  MoveL 9971 to (-27.77, 164.22, 135.08) mm, rotated rx 180 ry 0 rz 180 deg; joints [-126.617, -52.338, -80.882, 63.029, 64.237, -40.501]
  Call Extruder(390.70034)
  MoveL 9972 to (-28.02, 164.17, 135.08) mm, rotated rx 180 ry 0 rz 180 deg; joints [-126.595, -52.322, -80.919, 63.038, 64.26, -40.489]
  MoveL 9973 to (-28.02, 164.17, 135.08) mm, rotated rx 180 ry 0 rz 180 deg; joints [-126.595, -52.322, -80.919, 63.038, 64.26, -40.489]
  Call Extruder(390.83670)
  MoveL 9974 to (-28.27, 164.12, 135.08) mm, rotated rx 180 ry 0 rz -180 deg; joints [-126.573, -52.305, -80.957, 63.048, 64.284, -40.477]
  MoveL 9975 to (-28.27, 164.12, 135.08) mm, rotated rx 180 ry 0 rz -180 deg; joints [-126.573, -52.305, -80.957, 63.048, 64.284, -40.477]
  Call Extruder(390.97368)
  MoveL 9976 to (-28.52, 164.07, 135.08) mm, rotated rx 180 ry 0 rz 180 deg; joints [-126.551, -52.288, -80.994, 63.058, 64.307, -40.464]
  MoveL 9977 to (-28.52, 164.07, 135.08) mm, rotated rx 180 ry 0 rz 180 deg; joints [-126.551, -52.288, -80.994, 63.058, 64.307, -40.464]
  Call Extruder(391.11127)
  MoveL 9978 to (-28.77, 164.02, 135.08) mm, rotated rx -180 ry 0 rz 180 deg; joints [-126.529, -52.272, -81.031, 63.067, 64.331, -40.452]
  MoveL 9979 to (-28.77, 164.02, 135.08) mm, rotated rx -180 ry 0 rz 180 deg; joints [-126.529, -52.272, -81.031, 63.067, 64.331, -40.452]
  Call Extruder(391.22498)
  MoveL 9980 to (-28.97, 163.97, 135.08) mm, rotated rx 180 ry 0 rz 180 deg; joints [-126.511, -52.258, -81.062, 63.075, 64.35, -40.441]
  MoveL 9981 to (-28.97, 163.97, 135.08) mm, rotated rx 180 ry 0 rz 180 deg; joints [-126.511, -52.258, -81.062, 63.075, 64.35, -40.441]
  Call Extruder(391.33915)
  MoveL 9982 to (-29.18, 163.93, 135.08) mm, rotated rx 180 ry 0 rz 180 deg; joints [-126.494, -52.244, -81.093, 63.082, 64.369, -40.431]
  MoveL 9983 to (-29.18, 163.93, 135.08) mm, rotated rx 180 ry 0 rz 180 deg; joints [-126.494, -52.244, -81.093, 63.082, 64.369, -40.431]
  Call Extruder(391.45377)
  MoveL 9984 to (-29.38, 163.88, 135.08) mm, rotated rx -180 ry 0 rz 180 deg; joints [-126.476, -52.23, -81.125, 63.09, 64.389, -40.42]
  MoveL 9985 to (-29.38, 163.88, 135.08) mm, rotated rx -180 ry 0 rz 180 deg; joints [-126.476, -52.23, -81.125, 63.09, 64.389, -40.42]
  Call Extruder(391.56884)
  MoveL 9986 to (-29.59, 163.84, 135.08) mm, rotated rx 180 ry 0 rz 180 deg; joints [-126.459, -52.216, -81.155, 63.098, 64.408, -40.41]
  MoveL 9987 to (-29.59, 163.84, 135.08) mm, rotated rx 180 ry 0 rz 180 deg; joints [-126.459, -52.216, -81.155, 63.098, 64.408, -40.41]
  Call Extruder(391.69108)
  MoveL 9988 to (-29.8, 163.78, 135.08) mm, rotated rx -180 ry 0 rz 180 deg; joints [-126.441, -52.201, -81.189, 63.105, 64.428, -40.397]
  MoveL 9989 to (-29.8, 163.78, 135.08) mm, rotated rx -180 ry 0 rz 180 deg; joints [-126.441, -52.201, -81.189, 63.105, 64.428, -40.397]
  Call Extruder(391.82075)
  MoveL 9990 to (-30.02, 163.72, 135.08) mm, rotated rx -180 ry 0 rz 180 deg; joints [-126.423, -52.184, -81.227, 63.111, 64.449, -40.384]
  MoveL 9991 to (-30.02, 163.72, 135.08) mm, rotated rx -180 ry 0 rz 180 deg; joints [-126.423, -52.184, -81.227, 63.111, 64.449, -40.384]
  Call Extruder(391.95100)
  MoveL 9992 to (-30.25, 163.65, 135.08) mm, rotated rx 180 ry 0 rz 180 deg; joints [-126.405, -52.168, -81.263, 63.117, 64.47, -40.37]
  MoveL 9993 to (-30.25, 163.65, 135.08) mm, rotated rx 180 ry 0 rz 180 deg; joints [-126.405, -52.168, -81.263, 63.117, 64.47, -40.37]
  Call Extruder(392.08180)
  MoveL 9994 to (-30.47, 163.58, 135.08) mm, rotated rx 180 ry 0 rz 180 deg; joints [-126.387, -52.151, -81.3, 63.124, 64.491, -40.356]
  MoveL 9995 to (-30.47, 163.58, 135.08) mm, rotated rx 180 ry 0 rz 180 deg; joints [-126.387, -52.151, -81.3, 63.124, 64.491, -40.356]
  Call Extruder(392.21318)
  MoveL 9996 to (-30.69, 163.51, 135.08) mm, rotated rx 180 ry 0 rz 180 deg; joints [-126.369, -52.135, -81.337, 63.13, 64.512, -40.343]
  MoveL 9997 to (-30.69, 163.51, 135.08) mm, rotated rx 180 ry 0 rz 180 deg; joints [-126.369, -52.135, -81.337, 63.13, 64.512, -40.343]
  Call Extruder(392.32507)
  MoveL 9998 to (-30.88, 163.45, 135.08) mm, rotated rx 180 ry 0 rz 180 deg; joints [-126.354, -52.121, -81.369, 63.135, 64.529, -40.331]
  MoveL 9999 to (-30.88, 163.45, 135.08) mm, rotated rx 180 ry 0 rz 180 deg; joints [-126.354, -52.121, -81.369, 63.135, 64.529, -40.331]
  Call Extruder(392.43740)
  MoveL 10000 to (-31.07, 163.39, 135.08) mm, rotated rx 180 ry 0 rz 180 deg; joints [-126.339, -52.107, -81.401, 63.141, 64.547, -40.319]
  MoveL 10001 to (-31.07, 163.39, 135.08) mm, rotated rx 180 ry 0 rz 180 deg; joints [-126.339, -52.107, -81.401, 63.141, 64.547, -40.319]
  Call Extruder(392.55019)
  MoveL 10002 to (-31.26, 163.33, 135.08) mm, rotated rx 180 ry 0 rz 180 deg; joints [-126.324, -52.092, -81.433, 63.146, 64.564, -40.307]
  MoveL 10003 to (-31.26, 163.33, 135.08) mm, rotated rx 180 ry 0 rz 180 deg; joints [-126.324, -52.092, -81.433, 63.146, 64.564, -40.307]
  Call Extruder(392.66341)
  MoveL 10004 to (-31.45, 163.27, 135.08) mm, rotated rx -180 ry 0 rz -180 deg; joints [-126.309, -52.078, -81.464, 63.151, 64.582, -40.295]
  MoveL 10005 to (-31.45, 163.27, 135.08) mm, rotated rx -180 ry 0 rz -180 deg; joints [-126.309, -52.078, -81.464, 63.151, 64.582, -40.295]
  Call Extruder(392.77708)
  MoveL 10006 to (-31.64, 163.21, 135.08) mm, rotated rx 180 ry 0 rz 180 deg; joints [-126.294, -52.064, -81.496, 63.156, 64.599, -40.283]
  MoveL 10007 to (-31.64, 163.21, 135.08) mm, rotated rx 180 ry 0 rz 180 deg; joints [-126.294, -52.064, -81.496, 63.156, 64.599, -40.283]
  Call Extruder(392.95906)
  MoveL 10008 to (-31.93, 163.09, 135.08) mm, rotated rx 180 ry 0 rz 180 deg; joints [-126.273, -52.041, -81.549, 63.161, 64.626, -40.261]
  MoveL 10009 to (-31.93, 163.09, 135.08) mm, rotated rx 180 ry 0 rz 180 deg; joints [-126.273, -52.041, -81.549, 63.161, 64.626, -40.261]
  Call Extruder(393.14179)
  MoveL 10010 to (-32.22, 162.96, 135.08) mm, rotated rx -180 ry 0 rz -180 deg; joints [-126.252, -52.017, -81.602, 63.167, 64.653, -40.24]
  MoveL 10011 to (-32.22, 162.96, 135.08) mm, rotated rx -180 ry 0 rz -180 deg; joints [-126.252, -52.017, -81.602, 63.167, 64.653, -40.24]
  Call Extruder(393.31221)
  MoveL 10012 to (-32.49, 162.85, 135.08) mm, rotated rx 180 ry 0 rz -180 deg; joints [-126.233, -51.995, -81.652, 63.171, 64.678, -40.22]
  MoveL 10013 to (-32.49, 162.85, 135.08) mm, rotated rx 180 ry 0 rz -180 deg; joints [-126.233, -51.995, -81.652, 63.171, 64.678, -40.22]
  Call Extruder(393.47018)
  MoveL 10014 to (-32.74, 162.74, 135.08) mm, rotated rx -180 ry 0 rz 180 deg; joints [-126.215, -51.974, -81.698, 63.176, 64.701, -40.201]
  MoveL 10015 to (-32.74, 162.74, 135.08) mm, rotated rx -180 ry 0 rz 180 deg; joints [-126.215, -51.974, -81.698, 63.176, 64.701, -40.201]
  Call Extruder(393.62876)
  MoveL 10016 to (-32.99, 162.64, 135.08) mm, rotated rx 180 ry 0 rz 180 deg; joints [-126.197, -51.954, -81.744, 63.18, 64.724, -40.182]
  MoveL 10017 to (-32.99, 162.64, 135.08) mm, rotated rx 180 ry 0 rz 180 deg; joints [-126.197, -51.954, -81.744, 63.18, 64.724, -40.182]
  Call Extruder(393.83493)
  MoveL 10018 to (-33.29, 162.46, 135.08) mm, rotated rx 180 ry 0 rz 180 deg; joints [-126.179, -51.926, -81.807, 63.181, 64.752, -40.154]
  MoveL 10019 to (-33.29, 162.46, 135.08) mm, rotated rx 180 ry 0 rz 180 deg; joints [-126.179, -51.926, -81.807, 63.181, 64.752, -40.154]
  Call Extruder(394.04187)
  MoveL 10020 to (-33.6, 162.29, 135.08) mm, rotated rx 180 ry 0 rz -180 deg; joints [-126.16, -51.898, -81.87, 63.182, 64.78, -40.126]
  MoveL 10021 to (-33.6, 162.29, 135.08) mm, rotated rx 180 ry 0 rz -180 deg; joints [-126.16, -51.898, -81.87, 63.182, 64.78, -40.126]
  Call Extruder(394.24959)
  MoveL 10022 to (-33.9, 162.11, 135.08) mm, rotated rx 180 ry 0 rz -180 deg; joints [-126.142, -51.87, -81.933, 63.183, 64.807, -40.099]
  MoveL 10023 to (-33.9, 162.11, 135.08) mm, rotated rx 180 ry 0 rz -180 deg; joints [-126.142, -51.87, -81.933, 63.183, 64.807, -40.099]
  Call Extruder(394.45809)
  MoveL 10024 to (-34.21, 161.94, 135.08) mm, rotated rx 180 ry 0 rz -180 deg; joints [-126.123, -51.842, -81.996, 63.183, 64.835, -40.071]
  MoveL 10025 to (-34.21, 161.94, 135.08) mm, rotated rx 180 ry 0 rz -180 deg; joints [-126.123, -51.842, -81.996, 63.183, 64.835, -40.071]
  Call Extruder(394.63764)
  MoveL 10026 to (-34.45, 161.76, 135.08) mm, rotated rx 180 ry 0 rz 180 deg; joints [-126.111, -51.817, -82.052, 63.181, 64.857, -40.044]
  MoveL 10027 to (-34.45, 161.76, 135.08) mm, rotated rx 180 ry 0 rz 180 deg; joints [-126.111, -51.817, -82.052, 63.181, 64.857, -40.044]
  Call Extruder(394.97107)
  MoveL 10028 to (-34.9, 161.43, 135.08) mm, rotated rx 180 ry 0 rz 180 deg; joints [-126.089, -51.77, -82.156, 63.175, 64.897, -39.995]
  MoveL 10029 to (-34.9, 161.43, 135.08) mm, rotated rx 180 ry 0 rz 180 deg; joints [-126.089, -51.77, -82.156, 63.175, 64.897, -39.995]
  Call Extruder(395.30569)
  MoveL 10030 to (-35.35, 161.1, 135.08) mm, rotated rx 180 ry 0 rz 180 deg; joints [-126.067, -51.724, -82.26, 63.17, 64.938, -39.946]
  Call Extruder(396.13360)
  MoveL 10031 to (-36.39, 160.19, 135.08) mm, rotated rx 180 ry 0 rz 180 deg; joints [-126.027, -51.607, -82.524, 63.142, 65.029, -39.816]
  Call Extruder(396.96153)
  MoveL 10032 to (-37.3, 159.15, 135.08) mm, rotated rx -180 ry 0 rz 180 deg; joints [-126.011, -51.488, -82.792, 63.095, 65.107, -39.675]
  Call Extruder(397.12884)
  MoveL 10033 to (-37.47, 158.93, 135.08) mm, rotated rx 180 ry 0 rz 180 deg; joints [-126.011, -51.464, -82.846, 63.082, 65.121, -39.646]
  MoveL 10034 to (-37.47, 158.93, 135.08) mm, rotated rx 180 ry 0 rz 180 deg; joints [-126.011, -51.464, -82.846, 63.082, 65.121, -39.646]
  Call Extruder(397.46227)
  MoveL 10035 to (-37.79, 158.48, 135.08) mm, rotated rx -180 ry 0 rz -180 deg; joints [-126.011, -51.416, -82.955, 63.057, 65.148, -39.586]
  MoveL 10036 to (-37.79, 158.48, 135.08) mm, rotated rx -180 ry 0 rz -180 deg; joints [-126.011, -51.416, -82.955, 63.057, 65.148, -39.586]
  Call Extruder(397.53291)
  MoveL 10037 to (-37.87, 158.38, 135.08) mm, rotated rx 180 ry 0 rz 180 deg; joints [-126.011, -51.406, -82.978, 63.052, 65.154, -39.573]
  Set speed (130.0 mm/s)
  MoveL 10038 to (-39.48, 155.51, 135.08) mm, rotated rx -180 ry 0 rz 180 deg; joints [-126.062, -51.125, -83.613, 62.863, 65.283, -39.207]
  MoveL 10039 to (-39.48, 155.51, 144.49) mm, rotated rx 180 ry 0 rz 180 deg; joints [-126.062, -49.882, -84.026, 63.207, 64.906, -40.024]
  MoveL 10040 to (-38.84, 156.79, 144.49) mm, rotated rx 180 ry 0 rz 180 deg; joints [-126.03, -50.005, -83.751, 63.296, 64.858, -40.184]
  Set speed (30.0 mm/s)
  MoveL 10041 to (-38.84, 156.79, 144.49) mm, rotated rx 180 ry 0 rz 180 deg; joints [-126.03, -50.005, -83.751, 63.296, 64.858, -40.184]
  Call Extruder(397.61221)
  MoveL 10042 to (-38.89, 156.66, 144.49) mm, rotated rx 180 ry 0 rz 180 deg; joints [-126.034, -49.994, -83.777, 63.287, 64.862, -40.169]
  MoveL 10043 to (-38.89, 156.66, 144.49) mm, rotated rx 180 ry 0 rz 180 deg; joints [-126.034, -49.994, -83.777, 63.287, 64.862, -40.169]
  Call Extruder(397.77019)
  MoveL 10044 to (-39, 156.42, 144.49) mm, rotated rx 180 ry 0 rz 180 deg; joints [-126.042, -49.971, -83.828, 63.268, 64.87, -40.138]
  MoveL 10045 to (-39, 156.42, 144.49) mm, rotated rx 180 ry 0 rz 180 deg; joints [-126.042, -49.971, -83.828, 63.268, 64.87, -40.138]
  Call Extruder(397.92758)
  MoveL 10046 to (-39.1, 156.17, 144.49) mm, rotated rx 180 ry 0 rz -180 deg; joints [-126.05, -49.948, -83.88, 63.25, 64.877, -40.107]
  MoveL 10047 to (-39.1, 156.17, 144.49) mm, rotated rx 180 ry 0 rz -180 deg; joints [-126.05, -49.948, -83.88, 63.25, 64.877, -40.107]
  Call Extruder(398.11030)
  MoveL 10048 to (-39.23, 155.88, 144.49) mm, rotated rx 180 ry 0 rz 180 deg; joints [-126.06, -49.921, -83.939, 63.228, 64.886, -40.072]
  MoveL 10049 to (-39.23, 155.88, 144.49) mm, rotated rx 180 ry 0 rz 180 deg; joints [-126.06, -49.921, -83.939, 63.228, 64.886, -40.072]
  Call Extruder(398.29226)
  MoveL 10050 to (-39.35, 155.58, 144.49) mm, rotated rx 180 ry 0 rz 180 deg; joints [-126.07, -49.894, -83.999, 63.206, 64.894, -40.036]
  MoveL 10051 to (-39.35, 155.58, 144.49) mm, rotated rx 180 ry 0 rz 180 deg; joints [-126.07, -49.894, -83.999, 63.206, 64.894, -40.036]
  Call Extruder(398.43959)
  MoveL 10052 to (-39.44, 155.34, 144.49) mm, rotated rx 180 ry 0 rz -180 deg; joints [-126.079, -49.872, -84.047, 63.187, 64.9, -40.007]
  MoveL 10053 to (-39.44, 155.34, 144.49) mm, rotated rx 180 ry 0 rz -180 deg; joints [-126.079, -49.872, -84.047, 63.187, 64.9, -40.007]
  Call Extruder(398.55283)
  MoveL 10054 to (-39.5, 155.15, 144.49) mm, rotated rx 180 ry 0 rz 180 deg; joints [-126.087, -49.856, -84.083, 63.172, 64.904, -39.984]
  MoveL 10055 to (-39.5, 155.15, 144.49) mm, rotated rx 180 ry 0 rz 180 deg; joints [-126.087, -49.856, -84.083, 63.172, 64.904, -39.984]
  Call Extruder(398.66562)
  MoveL 10056 to (-39.56, 154.97, 144.49) mm, rotated rx 180 ry 0 rz 180 deg; joints [-126.095, -49.839, -84.119, 63.157, 64.908, -39.962]
  MoveL 10057 to (-39.56, 154.97, 144.49) mm, rotated rx 180 ry 0 rz 180 deg; joints [-126.095, -49.839, -84.119, 63.157, 64.908, -39.962]
  Call Extruder(398.77796)
  MoveL 10058 to (-39.62, 154.78, 144.49) mm, rotated rx 180 ry 0 rz 180 deg; joints [-126.103, -49.823, -84.156, 63.142, 64.912, -39.939]
  MoveL 10059 to (-39.62, 154.78, 144.49) mm, rotated rx 180 ry 0 rz 180 deg; joints [-126.103, -49.823, -84.156, 63.142, 64.912, -39.939]
  Call Extruder(398.88986)
  MoveL 10060 to (-39.68, 154.59, 144.49) mm, rotated rx -180 ry 0 rz 180 deg; joints [-126.111, -49.806, -84.192, 63.126, 64.915, -39.916]
  MoveL 10061 to (-39.68, 154.59, 144.49) mm, rotated rx -180 ry 0 rz 180 deg; joints [-126.111, -49.806, -84.192, 63.126, 64.915, -39.916]
  Call Extruder(399.01126)
  MoveL 10062 to (-39.75, 154.38, 144.49) mm, rotated rx 180 ry 0 rz 180 deg; joints [-126.12, -49.789, -84.232, 63.11, 64.919, -39.892]
  MoveL 10063 to (-39.75, 154.38, 144.49) mm, rotated rx 180 ry 0 rz 180 deg; joints [-126.12, -49.789, -84.232, 63.11, 64.919, -39.892]
  Call Extruder(399.14206)
  MoveL 10064 to (-39.81, 154.16, 144.49) mm, rotated rx -180 ry 0 rz 180 deg; joints [-126.131, -49.769, -84.275, 63.091, 64.924, -39.865]
  MoveL 10065 to (-39.81, 154.16, 144.49) mm, rotated rx -180 ry 0 rz 180 deg; joints [-126.131, -49.769, -84.275, 63.091, 64.924, -39.865]
  Call Extruder(399.27229)
  MoveL 10066 to (-39.88, 153.94, 144.49) mm, rotated rx 180 ry 0 rz 180 deg; joints [-126.141, -49.75, -84.317, 63.073, 64.928, -39.838]
  MoveL 10067 to (-39.88, 153.94, 144.49) mm, rotated rx 180 ry 0 rz 180 deg; joints [-126.141, -49.75, -84.317, 63.073, 64.928, -39.838]
  Call Extruder(399.40195)
  MoveL 10068 to (-39.95, 153.71, 144.49) mm, rotated rx -180 ry 0 rz 180 deg; joints [-126.151, -49.731, -84.36, 63.054, 64.932, -39.811]
  MoveL 10069 to (-39.95, 153.71, 144.49) mm, rotated rx -180 ry 0 rz 180 deg; joints [-126.151, -49.731, -84.36, 63.054, 64.932, -39.811]
  Call Extruder(399.53105)
  MoveL 10070 to (-40.02, 153.49, 144.49) mm, rotated rx -180 ry 0 rz -180 deg; joints [-126.161, -49.712, -84.402, 63.036, 64.936, -39.785]
  MoveL 10071 to (-40.02, 153.49, 144.49) mm, rotated rx -180 ry 0 rz -180 deg; joints [-126.161, -49.712, -84.402, 63.036, 64.936, -39.785]
  Call Extruder(399.64614)
  MoveL 10072 to (-40.06, 153.28, 144.49) mm, rotated rx -180 ry 0 rz 180 deg; joints [-126.173, -49.695, -84.439, 63.018, 64.938, -39.761]
  MoveL 10073 to (-40.06, 153.28, 144.49) mm, rotated rx -180 ry 0 rz 180 deg; joints [-126.173, -49.695, -84.439, 63.018, 64.938, -39.761]
  Call Extruder(399.76077)
  MoveL 10074 to (-40.11, 153.08, 144.49) mm, rotated rx 180 ry 0 rz -180 deg; joints [-126.184, -49.679, -84.476, 63, 64.94, -39.737]
  MoveL 10075 to (-40.11, 153.08, 144.49) mm, rotated rx 180 ry 0 rz -180 deg; joints [-126.184, -49.679, -84.476, 63, 64.94, -39.737]
  Call Extruder(399.87495)
  MoveL 10076 to (-40.15, 152.88, 144.49) mm, rotated rx -180 ry 0 rz -180 deg; joints [-126.195, -49.662, -84.513, 62.982, 64.942, -39.713]
  MoveL 10077 to (-40.15, 152.88, 144.49) mm, rotated rx -180 ry 0 rz -180 deg; joints [-126.195, -49.662, -84.513, 62.982, 64.942, -39.713]
  Call Extruder(399.98868)
  MoveL 10078 to (-40.2, 152.67, 144.49) mm, rotated rx -180 ry 0 rz 180 deg; joints [-126.206, -49.645, -84.55, 62.964, 64.944, -39.689]
  MoveL 10079 to (-40.2, 152.67, 144.49) mm, rotated rx -180 ry 0 rz 180 deg; joints [-126.206, -49.645, -84.55, 62.964, 64.944, -39.689]
  Call Extruder(400.11411)
  MoveL 10080 to (-40.24, 152.45, 144.49) mm, rotated rx 180 ry 0 rz 180 deg; joints [-126.219, -49.627, -84.59, 62.944, 64.946, -39.662]
  MoveL 10081 to (-40.24, 152.45, 144.49) mm, rotated rx 180 ry 0 rz 180 deg; joints [-126.219, -49.627, -84.59, 62.944, 64.946, -39.662]
  Call Extruder(400.25109)
  MoveL 10082 to (-40.29, 152.2, 144.49) mm, rotated rx 180 ry 0 rz 180 deg; joints [-126.233, -49.607, -84.635, 62.921, 64.948, -39.633]
  MoveL 10083 to (-40.29, 152.2, 144.49) mm, rotated rx 180 ry 0 rz 180 deg; joints [-126.233, -49.607, -84.635, 62.921, 64.948, -39.633]
  Call Extruder(400.38745)
  MoveL 10084 to (-40.34, 151.95, 144.49) mm, rotated rx 180 ry 0 rz 180 deg; joints [-126.248, -49.587, -84.679, 62.899, 64.95, -39.604]
  MoveL 10085 to (-40.34, 151.95, 144.49) mm, rotated rx 180 ry 0 rz 180 deg; joints [-126.248, -49.587, -84.679, 62.899, 64.95, -39.604]
  Call Extruder(400.52321)
  MoveL 10086 to (-40.39, 151.7, 144.49) mm, rotated rx 180 ry 0 rz 180 deg; joints [-126.262, -49.567, -84.724, 62.877, 64.952, -39.575]
  MoveL 10087 to (-40.39, 151.7, 144.49) mm, rotated rx 180 ry 0 rz 180 deg; joints [-126.262, -49.567, -84.724, 62.877, 64.952, -39.575]
  Call Extruder(400.65835)
  MoveL 10088 to (-40.44, 151.45, 144.49) mm, rotated rx 180 ry 0 rz 180 deg; joints [-126.276, -49.547, -84.768, 62.854, 64.954, -39.546]
  MoveL 10089 to (-40.44, 151.45, 144.49) mm, rotated rx 180 ry 0 rz 180 deg; joints [-126.276, -49.547, -84.768, 62.854, 64.954, -39.546]
  Call Extruder(400.79289)
  MoveL 10090 to (-40.49, 151.2, 144.49) mm, rotated rx 180 ry 0 rz 180 deg; joints [-126.291, -49.527, -84.812, 62.832, 64.956, -39.517]
  MoveL 10091 to (-40.49, 151.2, 144.49) mm, rotated rx 180 ry 0 rz 180 deg; joints [-126.291, -49.527, -84.812, 62.832, 64.956, -39.517]
  Call Extruder(400.92681)
  MoveL 10092 to (-40.54, 150.95, 144.49) mm, rotated rx 180 ry 0 rz -180 deg; joints [-126.305, -49.508, -84.856, 62.81, 64.958, -39.487]
  MoveL 10093 to (-40.54, 150.95, 144.49) mm, rotated rx 180 ry 0 rz -180 deg; joints [-126.305, -49.508, -84.856, 62.81, 64.958, -39.487]
  Call Extruder(401.07467)
  MoveL 10094 to (-40.59, 150.67, 144.49) mm, rotated rx 180 ry 0 rz -180 deg; joints [-126.322, -49.486, -84.905, 62.784, 64.959, -39.455]
  MoveL 10095 to (-40.59, 150.67, 144.49) mm, rotated rx 180 ry 0 rz -180 deg; joints [-126.322, -49.486, -84.905, 62.784, 64.959, -39.455]
  Call Extruder(401.23639)
  MoveL 10096 to (-40.64, 150.37, 144.49) mm, rotated rx -180 ry 0 rz 180 deg; joints [-126.341, -49.462, -84.958, 62.756, 64.961, -39.42]
  MoveL 10097 to (-40.64, 150.37, 144.49) mm, rotated rx -180 ry 0 rz 180 deg; joints [-126.341, -49.462, -84.958, 62.756, 64.961, -39.42]
  Call Extruder(401.39739)
  MoveL 10098 to (-40.69, 150.06, 144.49) mm, rotated rx 180 ry 0 rz -180 deg; joints [-126.36, -49.438, -85.011, 62.728, 64.962, -39.384]
  MoveL 10099 to (-40.69, 150.06, 144.49) mm, rotated rx 180 ry 0 rz -180 deg; joints [-126.36, -49.438, -85.011, 62.728, 64.962, -39.384]
  Call Extruder(401.55766)
  MoveL 10100 to (-40.74, 149.76, 144.49) mm, rotated rx 180 ry 0 rz 180 deg; joints [-126.379, -49.415, -85.063, 62.7, 64.963, -39.349]
  MoveL 10101 to (-40.74, 149.76, 144.49) mm, rotated rx 180 ry 0 rz 180 deg; joints [-126.379, -49.415, -85.063, 62.7, 64.963, -39.349]
  Call Extruder(401.71721)
  MoveL 10102 to (-40.78, 149.45, 144.49) mm, rotated rx 180 ry 0 rz -180 deg; joints [-126.398, -49.391, -85.116, 62.671, 64.964, -39.314]
  MoveL 10103 to (-40.78, 149.45, 144.49) mm, rotated rx 180 ry 0 rz -180 deg; joints [-126.398, -49.391, -85.116, 62.671, 64.964, -39.314]
  Call Extruder(401.87602)
  MoveL 10104 to (-40.83, 149.14, 144.49) mm, rotated rx 180 ry 0 rz 180 deg; joints [-126.417, -49.367, -85.169, 62.643, 64.966, -39.278]
  MoveL 10105 to (-40.83, 149.14, 144.49) mm, rotated rx 180 ry 0 rz 180 deg; joints [-126.417, -49.367, -85.169, 62.643, 64.966, -39.278]
  Call Extruder(402.05468)
  MoveL 10106 to (-40.88, 148.8, 144.49) mm, rotated rx 180 ry 0 rz 180 deg; joints [-126.439, -49.341, -85.228, 62.61, 64.966, -39.238]
  MoveL 10107 to (-40.88, 148.8, 144.49) mm, rotated rx 180 ry 0 rz 180 deg; joints [-126.439, -49.341, -85.228, 62.61, 64.966, -39.238]
  Call Extruder(402.25313)
  MoveL 10108 to (-40.92, 148.41, 144.49) mm, rotated rx 180 ry 0 rz 180 deg; joints [-126.465, -49.312, -85.293, 62.573, 64.966, -39.194]
  MoveL 10109 to (-40.92, 148.41, 144.49) mm, rotated rx 180 ry 0 rz 180 deg; joints [-126.465, -49.312, -85.293, 62.573, 64.966, -39.194]
  Call Extruder(402.45070)
  MoveL 10110 to (-40.97, 148.02, 144.49) mm, rotated rx -180 ry 0 rz -180 deg; joints [-126.491, -49.282, -85.358, 62.536, 64.967, -39.149]
  MoveL 10111 to (-40.97, 148.02, 144.49) mm, rotated rx -180 ry 0 rz -180 deg; joints [-126.491, -49.282, -85.358, 62.536, 64.967, -39.149]
  Call Extruder(402.64741)
  MoveL 10112 to (-41.02, 147.63, 144.49) mm, rotated rx -180 ry 0 rz 180 deg; joints [-126.517, -49.253, -85.423, 62.499, 64.967, -39.105]
  MoveL 10113 to (-41.02, 147.63, 144.49) mm, rotated rx -180 ry 0 rz 180 deg; joints [-126.517, -49.253, -85.423, 62.499, 64.967, -39.105]
  Call Extruder(402.84324)
  MoveL 10114 to (-41.06, 147.25, 144.49) mm, rotated rx -180 ry 0 rz 180 deg; joints [-126.543, -49.224, -85.487, 62.462, 64.967, -39.06]
  MoveL 10115 to (-41.06, 147.25, 144.49) mm, rotated rx -180 ry 0 rz 180 deg; joints [-126.543, -49.224, -85.487, 62.462, 64.967, -39.06]
  Call Extruder(403.13864)
  MoveL 10116 to (-41.11, 146.66, 144.49) mm, rotated rx -180 ry 0 rz 180 deg; joints [-126.585, -49.181, -85.583, 62.404, 64.965, -38.993]
  MoveL 10117 to (-41.11, 146.66, 144.49) mm, rotated rx -180 ry 0 rz 180 deg; joints [-126.585, -49.181, -85.583, 62.404, 64.965, -38.993]
  Call Extruder(403.43270)
  MoveL 10118 to (-41.15, 146.07, 144.49) mm, rotated rx -180 ry 0 rz 180 deg; joints [-126.628, -49.138, -85.679, 62.345, 64.962, -38.926]
  MoveL 10119 to (-41.15, 146.07, 144.49) mm, rotated rx -180 ry 0 rz 180 deg; joints [-126.628, -49.138, -85.679, 62.345, 64.962, -38.926]
  Call Extruder(403.72544)
  MoveL 10120 to (-41.2, 145.48, 144.49) mm, rotated rx 180 ry 0 rz 180 deg; joints [-126.67, -49.096, -85.775, 62.287, 64.96, -38.859]
  MoveL 10121 to (-41.2, 145.48, 144.49) mm, rotated rx 180 ry 0 rz 180 deg; joints [-126.67, -49.096, -85.775, 62.287, 64.96, -38.859]
  Call Extruder(404.29889)
  MoveL 10122 to (-41.25, 144.32, 144.49) mm, rotated rx 180 ry 0 rz 180 deg; joints [-126.759, -49.014, -85.958, 62.169, 64.952, -38.728]
  MoveL 10123 to (-41.25, 144.32, 144.49) mm, rotated rx 180 ry 0 rz 180 deg; joints [-126.759, -49.014, -85.958, 62.169, 64.952, -38.728]
  Call Extruder(405.01285)
  MoveL 10124 to (-41.29, 142.86, 144.49) mm, rotated rx -180 ry 0 rz 180 deg; joints [-126.873, -48.913, -86.184, 62.019, 64.939, -38.564]
  Call Extruder(447.07768)
  MoveL 10125 to (-41.29, 57.14, 144.49) mm, rotated rx 180 ry 0 rz 180 deg; joints [-135.148, -43.806, -97.993, 51.694, 63.997, -29.031]
  Call Extruder(447.50624)
  MoveL 10126 to (-41.27, 56.26, 144.49) mm, rotated rx 180 ry 0 rz 180 deg; joints [-135.25, -43.763, -98.098, 51.572, 63.986, -28.934]
  MoveL 10127 to (-41.27, 56.26, 144.49) mm, rotated rx 180 ry 0 rz 180 deg; joints [-135.25, -43.763, -98.098, 51.572, 63.986, -28.934]
  Call Extruder(448.07969)
  MoveL 10128 to (-41.22, 55.1, 144.49) mm, rotated rx 180 ry 0 rz 180 deg; joints [-135.387, -43.706, -98.235, 51.407, 63.969, -28.805]
  MoveL 10129 to (-41.22, 55.1, 144.49) mm, rotated rx 180 ry 0 rz 180 deg; joints [-135.387, -43.706, -98.235, 51.407, 63.969, -28.805]
  Call Extruder(448.51400)
  MoveL 10130 to (-41.18, 54.23, 144.49) mm, rotated rx 180 ry 0 rz 180 deg; joints [-135.493, -43.664, -98.337, 51.281, 63.956, -28.708]
  MoveL 10131 to (-41.18, 54.23, 144.49) mm, rotated rx 180 ry 0 rz 180 deg; joints [-135.493, -43.664, -98.337, 51.281, 63.956, -28.708]
  Call Extruder(448.80807)
  MoveL 10132 to (-41.13, 53.64, 144.49) mm, rotated rx 180 ry 0 rz 180 deg; joints [-135.566, -43.636, -98.403, 51.195, 63.945, -28.643]
  MoveL 10133 to (-41.13, 53.64, 144.49) mm, rotated rx 180 ry 0 rz 180 deg; joints [-135.566, -43.636, -98.403, 51.195, 63.945, -28.643]
  Call Extruder(449.10346)
  MoveL 10134 to (-41.09, 53.05, 144.49) mm, rotated rx -180 ry 0 rz -180 deg; joints [-135.64, -43.609, -98.469, 51.108, 63.934, -28.578]
  MoveL 10135 to (-41.09, 53.05, 144.49) mm, rotated rx -180 ry 0 rz -180 deg; joints [-135.64, -43.609, -98.469, 51.108, 63.934, -28.578]
  Call Extruder(449.34970)
  MoveL 10136 to (-41.04, 52.56, 144.49) mm, rotated rx 180 ry 0 rz -180 deg; joints [-135.701, -43.587, -98.523, 51.036, 63.924, -28.524]
  MoveL 10137 to (-41.04, 52.56, 144.49) mm, rotated rx 180 ry 0 rz -180 deg; joints [-135.701, -43.587, -98.523, 51.036, 63.924, -28.524]
  Call Extruder(449.54640)
  MoveL 10138 to (-40.99, 52.17, 144.49) mm, rotated rx 180 ry 0 rz 180 deg; joints [-135.751, -43.57, -98.564, 50.978, 63.916, -28.482]
  MoveL 10139 to (-40.99, 52.17, 144.49) mm, rotated rx 180 ry 0 rz 180 deg; joints [-135.751, -43.57, -98.564, 50.978, 63.916, -28.482]
  Call Extruder(449.74398)
  MoveL 10140 to (-40.95, 51.78, 144.49) mm, rotated rx 180 ry 0 rz 180 deg; joints [-135.801, -43.552, -98.605, 50.92, 63.907, -28.439]
  MoveL 10141 to (-40.95, 51.78, 144.49) mm, rotated rx 180 ry 0 rz 180 deg; joints [-135.801, -43.552, -98.605, 50.92, 63.907, -28.439]
  Call Extruder(449.94242)
  MoveL 10142 to (-40.9, 51.4, 144.49) mm, rotated rx -180 ry 0 rz -180 deg; joints [-135.852, -43.535, -98.647, 50.861, 63.898, -28.397]
  MoveL 10143 to (-40.9, 51.4, 144.49) mm, rotated rx -180 ry 0 rz -180 deg; joints [-135.852, -43.535, -98.647, 50.861, 63.898, -28.397]
  Call Extruder(450.14173)
  MoveL 10144 to (-40.86, 51.01, 144.49) mm, rotated rx 180 ry 0 rz -180 deg; joints [-135.902, -43.518, -98.688, 50.803, 63.89, -28.354]
  MoveL 10145 to (-40.86, 51.01, 144.49) mm, rotated rx 180 ry 0 rz -180 deg; joints [-135.902, -43.518, -98.688, 50.803, 63.89, -28.354]
  Call Extruder(450.30055)
  MoveL 10146 to (-40.81, 50.7, 144.49) mm, rotated rx -180 ry 0 rz -180 deg; joints [-135.943, -43.506, -98.719, 50.756, 63.882, -28.321]
  MoveL 10147 to (-40.81, 50.7, 144.49) mm, rotated rx -180 ry 0 rz -180 deg; joints [-135.943, -43.506, -98.719, 50.756, 63.882, -28.321]
  Call Extruder(450.46009)
  MoveL 10148 to (-40.76, 50.4, 144.49) mm, rotated rx 180 ry 0 rz -180 deg; joints [-135.984, -43.493, -98.749, 50.708, 63.874, -28.288]
  MoveL 10149 to (-40.76, 50.4, 144.49) mm, rotated rx 180 ry 0 rz -180 deg; joints [-135.984, -43.493, -98.749, 50.708, 63.874, -28.288]
  Call Extruder(450.62036)
  MoveL 10150 to (-40.71, 50.09, 144.49) mm, rotated rx -180 ry 0 rz -180 deg; joints [-136.025, -43.48, -98.78, 50.661, 63.866, -28.254]
  MoveL 10151 to (-40.71, 50.09, 144.49) mm, rotated rx -180 ry 0 rz -180 deg; joints [-136.025, -43.48, -98.78, 50.661, 63.866, -28.254]
  Call Extruder(450.78136)
  MoveL 10152 to (-40.66, 49.79, 144.49) mm, rotated rx 180 ry 0 rz -180 deg; joints [-136.067, -43.467, -98.811, 50.614, 63.858, -28.221]
  MoveL 10153 to (-40.66, 49.79, 144.49) mm, rotated rx 180 ry 0 rz -180 deg; joints [-136.067, -43.467, -98.811, 50.614, 63.858, -28.221]
  Call Extruder(450.94309)
  MoveL 10154 to (-40.61, 49.48, 144.49) mm, rotated rx 180 ry 0 rz -180 deg; joints [-136.108, -43.455, -98.842, 50.567, 63.85, -28.187]
  MoveL 10155 to (-40.61, 49.48, 144.49) mm, rotated rx 180 ry 0 rz -180 deg; joints [-136.108, -43.455, -98.842, 50.567, 63.85, -28.187]
  Call Extruder(451.10554)
  MoveL 10156 to (-40.57, 49.17, 144.49) mm, rotated rx -180 ry 0 rz 180 deg; joints [-136.149, -43.442, -98.873, 50.519, 63.842, -28.154]
  MoveL 10157 to (-40.57, 49.17, 144.49) mm, rotated rx -180 ry 0 rz 180 deg; joints [-136.149, -43.442, -98.873, 50.519, 63.842, -28.154]
  Call Extruder(451.23946)
  MoveL 10158 to (-40.52, 48.93, 144.49) mm, rotated rx 180 ry 0 rz 180 deg; joints [-136.184, -43.432, -98.896, 50.48, 63.834, -28.127]
  MoveL 10159 to (-40.52, 48.93, 144.49) mm, rotated rx 180 ry 0 rz 180 deg; joints [-136.184, -43.432, -98.896, 50.48, 63.834, -28.127]
  Call Extruder(451.37400)
  MoveL 10160 to (-40.47, 48.68, 144.49) mm, rotated rx -180 ry 0 rz 180 deg; joints [-136.219, -43.422, -98.92, 50.44, 63.827, -28.1]
  MoveL 10161 to (-40.47, 48.68, 144.49) mm, rotated rx -180 ry 0 rz 180 deg; joints [-136.219, -43.422, -98.92, 50.44, 63.827, -28.1]
  Call Extruder(451.50914)
  MoveL 10162 to (-40.42, 48.43, 144.49) mm, rotated rx 180 ry 0 rz -180 deg; joints [-136.254, -43.413, -98.944, 50.401, 63.819, -28.073]
  MoveL 10163 to (-40.42, 48.43, 144.49) mm, rotated rx 180 ry 0 rz -180 deg; joints [-136.254, -43.413, -98.944, 50.401, 63.819, -28.073]
  Call Extruder(451.64490)
  MoveL 10164 to (-40.37, 48.18, 144.49) mm, rotated rx 180 ry 0 rz 180 deg; joints [-136.288, -43.403, -98.967, 50.361, 63.811, -28.046]
  MoveL 10165 to (-40.37, 48.18, 144.49) mm, rotated rx 180 ry 0 rz 180 deg; joints [-136.288, -43.403, -98.967, 50.361, 63.811, -28.046]
  Call Extruder(451.78127)
  MoveL 10166 to (-40.32, 47.93, 144.49) mm, rotated rx 180 ry 0 rz -180 deg; joints [-136.323, -43.393, -98.991, 50.321, 63.804, -28.019]
  MoveL 10167 to (-40.32, 47.93, 144.49) mm, rotated rx 180 ry 0 rz -180 deg; joints [-136.323, -43.393, -98.991, 50.321, 63.804, -28.019]
  Call Extruder(451.91824)
  MoveL 10168 to (-40.27, 47.68, 144.49) mm, rotated rx -180 ry 0 rz 180 deg; joints [-136.358, -43.383, -99.015, 50.282, 63.796, -27.992]
  MoveL 10169 to (-40.27, 47.68, 144.49) mm, rotated rx -180 ry 0 rz 180 deg; joints [-136.358, -43.383, -99.015, 50.282, 63.796, -27.992]
  Call Extruder(452.05583)
  MoveL 10170 to (-40.22, 47.43, 144.49) mm, rotated rx 180 ry 0 rz 180 deg; joints [-136.393, -43.374, -99.038, 50.242, 63.789, -27.965]
  MoveL 10171 to (-40.22, 47.43, 144.49) mm, rotated rx 180 ry 0 rz 180 deg; joints [-136.393, -43.374, -99.038, 50.242, 63.789, -27.965]
  Call Extruder(452.16955)
  MoveL 10172 to (-40.17, 47.23, 144.49) mm, rotated rx -180 ry 0 rz -180 deg; joints [-136.422, -43.366, -99.057, 50.209, 63.782, -27.942]
  MoveL 10173 to (-40.17, 47.23, 144.49) mm, rotated rx -180 ry 0 rz -180 deg; joints [-136.422, -43.366, -99.057, 50.209, 63.782, -27.942]
  Call Extruder(452.28373)
  MoveL 10174 to (-40.13, 47.02, 144.49) mm, rotated rx 180 ry 0 rz 180 deg; joints [-136.452, -43.358, -99.076, 50.176, 63.776, -27.92]
  MoveL 10175 to (-40.13, 47.02, 144.49) mm, rotated rx 180 ry 0 rz 180 deg; joints [-136.452, -43.358, -99.076, 50.176, 63.776, -27.92]
  Call Extruder(452.39837)
  MoveL 10176 to (-40.08, 46.82, 144.49) mm, rotated rx -180 ry 0 rz -180 deg; joints [-136.481, -43.35, -99.095, 50.143, 63.769, -27.898]
  MoveL 10177 to (-40.08, 46.82, 144.49) mm, rotated rx -180 ry 0 rz -180 deg; joints [-136.481, -43.35, -99.095, 50.143, 63.769, -27.898]
  Call Extruder(452.51345)
  MoveL 10178 to (-40.04, 46.61, 144.49) mm, rotated rx 180 ry 0 rz 180 deg; joints [-136.51, -43.343, -99.113, 50.111, 63.763, -27.876]
  MoveL 10179 to (-40.04, 46.61, 144.49) mm, rotated rx 180 ry 0 rz 180 deg; joints [-136.51, -43.343, -99.113, 50.111, 63.763, -27.876]
  Call Extruder(452.63569)
  MoveL 10180 to (-39.98, 46.4, 144.49) mm, rotated rx 180 ry 0 rz -180 deg; joints [-136.542, -43.335, -99.132, 50.075, 63.755, -27.853]
  MoveL 10181 to (-39.98, 46.4, 144.49) mm, rotated rx 180 ry 0 rz -180 deg; joints [-136.542, -43.335, -99.132, 50.075, 63.755, -27.853]
  Call Extruder(452.76536)
  MoveL 10182 to (-39.92, 46.18, 144.49) mm, rotated rx -180 ry 0 rz 180 deg; joints [-136.576, -43.328, -99.15, 50.037, 63.746, -27.829]
  MoveL 10183 to (-39.92, 46.18, 144.49) mm, rotated rx -180 ry 0 rz 180 deg; joints [-136.576, -43.328, -99.15, 50.037, 63.746, -27.829]
  Call Extruder(452.89558)
  MoveL 10184 to (-39.85, 45.95, 144.49) mm, rotated rx -180 ry 0 rz 180 deg; joints [-136.61, -43.32, -99.168, 50, 63.736, -27.805]
  MoveL 10185 to (-39.85, 45.95, 144.49) mm, rotated rx -180 ry 0 rz 180 deg; joints [-136.61, -43.32, -99.168, 50, 63.736, -27.805]
  Call Extruder(453.02638)
  MoveL 10186 to (-39.78, 45.73, 144.49) mm, rotated rx 180 ry 0 rz 180 deg; joints [-136.644, -43.313, -99.186, 49.962, 63.727, -27.781]
  MoveL 10187 to (-39.78, 45.73, 144.49) mm, rotated rx 180 ry 0 rz 180 deg; joints [-136.644, -43.313, -99.186, 49.962, 63.727, -27.781]
  Call Extruder(453.15773)
  MoveL 10188 to (-39.71, 45.5, 144.49) mm, rotated rx -180 ry 0 rz -180 deg; joints [-136.678, -43.305, -99.204, 49.924, 63.718, -27.757]
  MoveL 10189 to (-39.71, 45.5, 144.49) mm, rotated rx -180 ry 0 rz -180 deg; joints [-136.678, -43.305, -99.204, 49.924, 63.718, -27.757]
  Call Extruder(453.26964)
  MoveL 10190 to (-39.65, 45.32, 144.49) mm, rotated rx -180 ry 0 rz -180 deg; joints [-136.707, -43.299, -99.219, 49.892, 63.71, -27.737]
  MoveL 10191 to (-39.65, 45.32, 144.49) mm, rotated rx -180 ry 0 rz -180 deg; joints [-136.707, -43.299, -99.219, 49.892, 63.71, -27.737]
  Call Extruder(453.38198)
  MoveL 10192 to (-39.59, 45.13, 144.49) mm, rotated rx 180 ry 0 rz 180 deg; joints [-136.737, -43.293, -99.234, 49.86, 63.702, -27.716]
  MoveL 10193 to (-39.59, 45.13, 144.49) mm, rotated rx 180 ry 0 rz 180 deg; joints [-136.737, -43.293, -99.234, 49.86, 63.702, -27.716]
  Call Extruder(453.49477)
  MoveL 10194 to (-39.53, 44.94, 144.49) mm, rotated rx 180 ry 0 rz 180 deg; joints [-136.766, -43.287, -99.248, 49.828, 63.694, -27.696]
  MoveL 10195 to (-39.53, 44.94, 144.49) mm, rotated rx 180 ry 0 rz 180 deg; joints [-136.766, -43.287, -99.248, 49.828, 63.694, -27.696]
  Call Extruder(453.60801)
  MoveL 10196 to (-39.47, 44.75, 144.49) mm, rotated rx 180 ry 0 rz -180 deg; joints [-136.796, -43.281, -99.263, 49.795, 63.686, -27.676]
  MoveL 10197 to (-39.47, 44.75, 144.49) mm, rotated rx 180 ry 0 rz -180 deg; joints [-136.796, -43.281, -99.263, 49.795, 63.686, -27.676]
  Call Extruder(453.72169)
  MoveL 10198 to (-39.41, 44.56, 144.49) mm, rotated rx 180 ry 0 rz -180 deg; joints [-136.825, -43.275, -99.278, 49.763, 63.678, -27.656]
  MoveL 10199 to (-39.41, 44.56, 144.49) mm, rotated rx 180 ry 0 rz -180 deg; joints [-136.825, -43.275, -99.278, 49.763, 63.678, -27.656]
  Call Extruder(453.90365)
  MoveL 10200 to (-39.29, 44.27, 144.49) mm, rotated rx 180 ry 0 rz -180 deg; joints [-136.873, -43.267, -99.297, 49.711, 63.663, -27.625]
  MoveL 10201 to (-39.29, 44.27, 144.49) mm, rotated rx 180 ry 0 rz -180 deg; joints [-136.873, -43.267, -99.297, 49.711, 63.663, -27.625]
  Call Extruder(454.08636)
  MoveL 10202 to (-39.16, 43.98, 144.49) mm, rotated rx -180 ry 0 rz 180 deg; joints [-136.922, -43.259, -99.316, 49.659, 63.648, -27.594]
  MoveL 10203 to (-39.16, 43.98, 144.49) mm, rotated rx -180 ry 0 rz 180 deg; joints [-136.922, -43.259, -99.316, 49.659, 63.648, -27.594]
  Call Extruder(454.25678)
  MoveL 10204 to (-39.05, 43.71, 144.49) mm, rotated rx 180 ry 0 rz 180 deg; joints [-136.967, -43.252, -99.334, 49.61, 63.634, -27.565]
  MoveL 10205 to (-39.05, 43.71, 144.49) mm, rotated rx 180 ry 0 rz 180 deg; joints [-136.967, -43.252, -99.334, 49.61, 63.634, -27.565]
  Call Extruder(454.41476)
  MoveL 10206 to (-38.94, 43.46, 144.49) mm, rotated rx 180 ry 0 rz 180 deg; joints [-137.009, -43.246, -99.35, 49.566, 63.62, -27.539]
  MoveL 10207 to (-38.94, 43.46, 144.49) mm, rotated rx 180 ry 0 rz 180 deg; joints [-137.009, -43.246, -99.35, 49.566, 63.62, -27.539]
  Call Extruder(454.57335)
  MoveL 10208 to (-38.84, 43.21, 144.49) mm, rotated rx 180 ry 0 rz 180 deg; joints [-137.05, -43.239, -99.365, 49.52, 63.607, -27.513]
  MoveL 10209 to (-38.84, 43.21, 144.49) mm, rotated rx 180 ry 0 rz 180 deg; joints [-137.05, -43.239, -99.365, 49.52, 63.607, -27.513]
  Call Extruder(454.77952)
  MoveL 10210 to (-38.66, 42.91, 144.49) mm, rotated rx 180 ry 0 rz -180 deg; joints [-137.107, -43.233, -99.379, 49.462, 63.586, -27.481]
  MoveL 10211 to (-38.66, 42.91, 144.49) mm, rotated rx 180 ry 0 rz -180 deg; joints [-137.107, -43.233, -99.379, 49.462, 63.586, -27.481]
  Call Extruder(454.98646)
  MoveL 10212 to (-38.49, 42.6, 144.49) mm, rotated rx -180 ry 0 rz 180 deg; joints [-137.163, -43.228, -99.393, 49.403, 63.566, -27.45]
  MoveL 10213 to (-38.49, 42.6, 144.49) mm, rotated rx -180 ry 0 rz 180 deg; joints [-137.163, -43.228, -99.393, 49.403, 63.566, -27.45]
  Call Extruder(455.19419)
  MoveL 10214 to (-38.31, 42.3, 144.49) mm, rotated rx 180 ry 0 rz 180 deg; joints [-137.219, -43.222, -99.406, 49.345, 63.545, -27.418]
  MoveL 10215 to (-38.31, 42.3, 144.49) mm, rotated rx 180 ry 0 rz 180 deg; joints [-137.219, -43.222, -99.406, 49.345, 63.545, -27.418]
  Call Extruder(455.40269)
  MoveL 10216 to (-38.14, 41.99, 144.49) mm, rotated rx -180 ry 0 rz 180 deg; joints [-137.275, -43.217, -99.419, 49.286, 63.524, -27.387]
  MoveL 10217 to (-38.14, 41.99, 144.49) mm, rotated rx -180 ry 0 rz 180 deg; joints [-137.275, -43.217, -99.419, 49.286, 63.524, -27.387]
  Call Extruder(455.58224)
  MoveL 10218 to (-37.96, 41.75, 144.49) mm, rotated rx 180 ry 0 rz -180 deg; joints [-137.324, -43.214, -99.426, 49.236, 63.504, -27.362]
  MoveL 10219 to (-37.96, 41.75, 144.49) mm, rotated rx 180 ry 0 rz -180 deg; joints [-137.324, -43.214, -99.426, 49.236, 63.504, -27.362]
  Call Extruder(455.91567)
  MoveL 10220 to (-37.63, 41.3, 144.49) mm, rotated rx -180 ry 0 rz 180 deg; joints [-137.415, -43.21, -99.437, 49.143, 63.467, -27.316]
  MoveL 10221 to (-37.63, 41.3, 144.49) mm, rotated rx -180 ry 0 rz 180 deg; joints [-137.415, -43.21, -99.437, 49.143, 63.467, -27.316]
  Call Extruder(456.25030)
  MoveL 10222 to (-37.3, 40.85, 144.49) mm, rotated rx 180 ry 0 rz 180 deg; joints [-137.506, -43.205, -99.448, 49.05, 63.429, -27.27]
  Call Extruder(457.07823)
  MoveL 10223 to (-36.39, 39.81, 144.49) mm, rotated rx 180 ry 0 rz -180 deg; joints [-137.733, -43.203, -99.452, 48.824, 63.327, -27.167]
  Call Extruder(457.90614)
  MoveL 10224 to (-35.35, 38.9, 144.49) mm, rotated rx 180 ry 0 rz -180 deg; joints [-137.958, -43.214, -99.425, 48.605, 63.214, -27.079]
  Call Extruder(458.07344)
  MoveL 10225 to (-35.13, 38.73, 144.49) mm, rotated rx 180 ry 0 rz 180 deg; joints [-138.003, -43.219, -99.415, 48.563, 63.19, -27.064]
  MoveL 10226 to (-35.13, 38.73, 144.49) mm, rotated rx 180 ry 0 rz 180 deg; joints [-138.003, -43.219, -99.415, 48.563, 63.19, -27.064]
  Call Extruder(458.40687)
  MoveL 10227 to (-34.68, 38.41, 144.49) mm, rotated rx 180 ry 0 rz 180 deg; joints [-138.092, -43.227, -99.395, 48.478, 63.141, -27.034]
  MoveL 10228 to (-34.68, 38.41, 144.49) mm, rotated rx 180 ry 0 rz 180 deg; joints [-138.092, -43.227, -99.395, 48.478, 63.141, -27.034]
  Call Extruder(458.73911)
  MoveL 10229 to (-34.22, 38.08, 144.49) mm, rotated rx 180 ry 0 rz -180 deg; joints [-138.182, -43.235, -99.375, 48.393, 63.092, -27.003]
  MoveL 10230 to (-34.22, 38.08, 144.49) mm, rotated rx 180 ry 0 rz -180 deg; joints [-138.182, -43.235, -99.375, 48.393, 63.092, -27.003]
  Call Extruder(458.85681)
  MoveL 10231 to (-34.05, 37.98, 144.49) mm, rotated rx 180 ry 0 rz 180 deg; joints [-138.213, -43.24, -99.364, 48.365, 63.074, -26.995]
  MoveL 10232 to (-34.05, 37.98, 144.49) mm, rotated rx 180 ry 0 rz 180 deg; joints [-138.213, -43.24, -99.364, 48.365, 63.074, -26.995]
  Call Extruder(459.06453)
  MoveL 10233 to (-33.75, 37.8, 144.49) mm, rotated rx -180 ry 0 rz 180 deg; joints [-138.267, -43.247, -99.345, 48.314, 63.042, -26.979]
  MoveL 10234 to (-33.75, 37.8, 144.49) mm, rotated rx -180 ry 0 rz 180 deg; joints [-138.267, -43.247, -99.345, 48.314, 63.042, -26.979]
  Call Extruder(459.27147)
  MoveL 10235 to (-33.45, 37.63, 144.49) mm, rotated rx -180 ry 0 rz -180 deg; joints [-138.322, -43.255, -99.326, 48.264, 63.01, -26.964]
  MoveL 10236 to (-33.45, 37.63, 144.49) mm, rotated rx -180 ry 0 rz -180 deg; joints [-138.322, -43.255, -99.326, 48.264, 63.01, -26.964]
  Call Extruder(459.47764)
  MoveL 10237 to (-33.14, 37.45, 144.49) mm, rotated rx -180 ry 0 rz -180 deg; joints [-138.376, -43.263, -99.307, 48.214, 62.978, -26.949]
  MoveL 10238 to (-33.14, 37.45, 144.49) mm, rotated rx -180 ry 0 rz -180 deg; joints [-138.376, -43.263, -99.307, 48.214, 62.978, -26.949]
  Call Extruder(459.65932)
  MoveL 10239 to (-32.87, 37.31, 144.49) mm, rotated rx 180 ry 0 rz 180 deg; joints [-138.424, -43.271, -99.287, 48.171, 62.948, -26.937]
  MoveL 10240 to (-32.87, 37.31, 144.49) mm, rotated rx 180 ry 0 rz 180 deg; joints [-138.424, -43.271, -99.287, 48.171, 62.948, -26.937]
  Call Extruder(459.81731)
  MoveL 10241 to (-32.62, 37.2, 144.49) mm, rotated rx -180 ry 0 rz -180 deg; joints [-138.464, -43.279, -99.267, 48.135, 62.922, -26.928]
  MoveL 10242 to (-32.62, 37.2, 144.49) mm, rotated rx -180 ry 0 rz -180 deg; joints [-138.464, -43.279, -99.267, 48.135, 62.922, -26.928]
  Call Extruder(459.97470)
  MoveL 10243 to (-32.37, 37.1, 144.49) mm, rotated rx 180 ry 0 rz -180 deg; joints [-138.504, -43.288, -99.247, 48.099, 62.896, -26.92]
  MoveL 10244 to (-32.37, 37.1, 144.49) mm, rotated rx 180 ry 0 rz -180 deg; joints [-138.504, -43.288, -99.247, 48.099, 62.896, -26.92]
  Call Extruder(460.13371)
  MoveL 10245 to (-32.11, 36.99, 144.49) mm, rotated rx 180 ry 0 rz 180 deg; joints [-138.545, -43.296, -99.226, 48.063, 62.87, -26.912]
  MoveL 10246 to (-32.11, 36.99, 144.49) mm, rotated rx 180 ry 0 rz 180 deg; joints [-138.545, -43.296, -99.226, 48.063, 62.87, -26.912]
  Call Extruder(460.28213)
  MoveL 10247 to (-31.87, 36.89, 144.49) mm, rotated rx 180 ry 0 rz -180 deg; joints [-138.582, -43.304, -99.207, 48.03, 62.845, -26.904]
  MoveL 10248 to (-31.87, 36.89, 144.49) mm, rotated rx 180 ry 0 rz -180 deg; joints [-138.582, -43.304, -99.207, 48.03, 62.845, -26.904]
  Call Extruder(460.43006)
  MoveL 10249 to (-31.64, 36.79, 144.49) mm, rotated rx 180 ry 0 rz 180 deg; joints [-138.62, -43.312, -99.187, 47.996, 62.82, -26.896]
  MoveL 10250 to (-31.64, 36.79, 144.49) mm, rotated rx 180 ry 0 rz 180 deg; joints [-138.62, -43.312, -99.187, 47.996, 62.82, -26.896]
  Call Extruder(460.54351)
  MoveL 10251 to (-31.45, 36.73, 144.49) mm, rotated rx 180 ry 0 rz -180 deg; joints [-138.648, -43.32, -99.17, 47.972, 62.801, -26.892]
  MoveL 10252 to (-31.45, 36.73, 144.49) mm, rotated rx 180 ry 0 rz -180 deg; joints [-138.648, -43.32, -99.17, 47.972, 62.801, -26.892]
  Call Extruder(460.65653)
  MoveL 10253 to (-31.26, 36.67, 144.49) mm, rotated rx 180 ry 0 rz 180 deg; joints [-138.676, -43.327, -99.152, 47.948, 62.781, -26.888]
  MoveL 10254 to (-31.26, 36.67, 144.49) mm, rotated rx 180 ry 0 rz 180 deg; joints [-138.676, -43.327, -99.152, 47.948, 62.781, -26.888]
  Call Extruder(460.76910)
  MoveL 10255 to (-31.07, 36.61, 144.49) mm, rotated rx 180 ry 0 rz -180 deg; joints [-138.704, -43.334, -99.135, 47.924, 62.762, -26.884]
  MoveL 10256 to (-31.07, 36.61, 144.49) mm, rotated rx 180 ry 0 rz -180 deg; joints [-138.704, -43.334, -99.135, 47.924, 62.762, -26.884]
  Call Extruder(460.88122)
  MoveL 10257 to (-30.88, 36.55, 144.49) mm, rotated rx -180 ry 0 rz -180 deg; joints [-138.732, -43.341, -99.117, 47.9, 62.742, -26.88]
  MoveL 10258 to (-30.88, 36.55, 144.49) mm, rotated rx -180 ry 0 rz -180 deg; joints [-138.732, -43.341, -99.117, 47.9, 62.742, -26.88]
  Call Extruder(460.99290)
  MoveL 10259 to (-30.69, 36.49, 144.49) mm, rotated rx 180 ry 0 rz -180 deg; joints [-138.759, -43.348, -99.1, 47.877, 62.723, -26.875]
  MoveL 10260 to (-30.69, 36.49, 144.49) mm, rotated rx 180 ry 0 rz -180 deg; joints [-138.759, -43.348, -99.1, 47.877, 62.723, -26.875]
  Call Extruder(461.12397)
  MoveL 10261 to (-30.47, 36.42, 144.49) mm, rotated rx 180 ry 0 rz 180 deg; joints [-138.792, -43.357, -99.078, 47.849, 62.7, -26.871]
  MoveL 10262 to (-30.47, 36.42, 144.49) mm, rotated rx 180 ry 0 rz 180 deg; joints [-138.792, -43.357, -99.078, 47.849, 62.7, -26.871]
  Call Extruder(461.25448)
  MoveL 10263 to (-30.25, 36.35, 144.49) mm, rotated rx 180 ry 0 rz -180 deg; joints [-138.824, -43.366, -99.056, 47.821, 62.676, -26.867]
  MoveL 10264 to (-30.25, 36.35, 144.49) mm, rotated rx 180 ry 0 rz -180 deg; joints [-138.824, -43.366, -99.056, 47.821, 62.676, -26.867]
  Call Extruder(461.38443)
  MoveL 10265 to (-30.02, 36.28, 144.49) mm, rotated rx 180 ry 0 rz -180 deg; joints [-138.856, -43.375, -99.035, 47.794, 62.653, -26.862]
  MoveL 10266 to (-30.02, 36.28, 144.49) mm, rotated rx 180 ry 0 rz -180 deg; joints [-138.856, -43.375, -99.035, 47.794, 62.653, -26.862]
  Call Extruder(461.51381)
  MoveL 10267 to (-29.8, 36.22, 144.49) mm, rotated rx 180 ry 0 rz -180 deg; joints [-138.889, -43.384, -99.014, 47.766, 62.63, -26.858]
  MoveL 10268 to (-29.8, 36.22, 144.49) mm, rotated rx 180 ry 0 rz -180 deg; joints [-138.889, -43.384, -99.014, 47.766, 62.63, -26.858]
  Call Extruder(461.63577)
  MoveL 10269 to (-29.59, 36.16, 144.49) mm, rotated rx -180 ry 0 rz -180 deg; joints [-138.919, -43.393, -98.992, 47.741, 62.608, -26.855]
  MoveL 10270 to (-29.59, 36.16, 144.49) mm, rotated rx -180 ry 0 rz -180 deg; joints [-138.919, -43.393, -98.992, 47.741, 62.608, -26.855]
  Call Extruder(461.75062)
  MoveL 10271 to (-29.38, 36.12, 144.49) mm, rotated rx -180 ry 0 rz -180 deg; joints [-138.946, -43.402, -98.97, 47.718, 62.587, -26.853]
  MoveL 10272 to (-29.38, 36.12, 144.49) mm, rotated rx -180 ry 0 rz -180 deg; joints [-138.946, -43.402, -98.97, 47.718, 62.587, -26.853]
  Call Extruder(461.86501)
  MoveL 10273 to (-29.18, 36.07, 144.49) mm, rotated rx 180 ry 0 rz 180 deg; joints [-138.973, -43.411, -98.949, 47.696, 62.566, -26.851]
  MoveL 10274 to (-29.18, 36.07, 144.49) mm, rotated rx 180 ry 0 rz 180 deg; joints [-138.973, -43.411, -98.949, 47.696, 62.566, -26.851]
  Call Extruder(461.97895)
  MoveL 10275 to (-28.97, 36.03, 144.49) mm, rotated rx 180 ry 0 rz -180 deg; joints [-139, -43.419, -98.927, 47.673, 62.546, -26.849]
  MoveL 10276 to (-28.97, 36.03, 144.49) mm, rotated rx 180 ry 0 rz -180 deg; joints [-139, -43.419, -98.927, 47.673, 62.546, -26.849]
  Call Extruder(462.09244)
  MoveL 10277 to (-28.77, 35.98, 144.49) mm, rotated rx 180 ry 0 rz -180 deg; joints [-139.028, -43.428, -98.905, 47.651, 62.525, -26.847]
  MoveL 10278 to (-28.77, 35.98, 144.49) mm, rotated rx 180 ry 0 rz -180 deg; joints [-139.028, -43.428, -98.905, 47.651, 62.525, -26.847]
  Call Extruder(462.22973)
  MoveL 10279 to (-28.52, 35.93, 144.49) mm, rotated rx -180 ry 0 rz 180 deg; joints [-139.06, -43.44, -98.878, 47.624, 62.499, -26.845]
  MoveL 10280 to (-28.52, 35.93, 144.49) mm, rotated rx -180 ry 0 rz 180 deg; joints [-139.06, -43.44, -98.878, 47.624, 62.499, -26.845]
  Call Extruder(462.36640)
  MoveL 10281 to (-28.27, 35.88, 144.49) mm, rotated rx -180 ry 0 rz 180 deg; joints [-139.093, -43.451, -98.851, 47.597, 62.474, -26.843]
  MoveL 10282 to (-28.27, 35.88, 144.49) mm, rotated rx -180 ry 0 rz 180 deg; joints [-139.093, -43.451, -98.851, 47.597, 62.474, -26.843]
  Call Extruder(462.50246)
  MoveL 10283 to (-28.02, 35.83, 144.49) mm, rotated rx 180 ry 0 rz 180 deg; joints [-139.126, -43.462, -98.824, 47.571, 62.448, -26.841]
  MoveL 10284 to (-28.02, 35.83, 144.49) mm, rotated rx 180 ry 0 rz 180 deg; joints [-139.126, -43.462, -98.824, 47.571, 62.448, -26.841]
  Call Extruder(462.63791)
  MoveL 10285 to (-27.77, 35.78, 144.49) mm, rotated rx 180 ry 0 rz 180 deg; joints [-139.158, -43.473, -98.797, 47.544, 62.423, -26.839]
  MoveL 10286 to (-27.77, 35.78, 144.49) mm, rotated rx 180 ry 0 rz 180 deg; joints [-139.158, -43.473, -98.797, 47.544, 62.423, -26.839]
  Call Extruder(462.77275)
  MoveL 10287 to (-27.52, 35.73, 144.49) mm, rotated rx 180 ry 0 rz 180 deg; joints [-139.191, -43.484, -98.77, 47.517, 62.398, -26.837]
  MoveL 10288 to (-27.52, 35.73, 144.49) mm, rotated rx 180 ry 0 rz 180 deg; joints [-139.191, -43.484, -98.77, 47.517, 62.398, -26.837]
  Call Extruder(462.90698)
  MoveL 10289 to (-27.28, 35.68, 144.49) mm, rotated rx -180 ry 0 rz -180 deg; joints [-139.223, -43.496, -98.743, 47.491, 62.372, -26.835]
  MoveL 10290 to (-27.28, 35.68, 144.49) mm, rotated rx -180 ry 0 rz -180 deg; joints [-139.223, -43.496, -98.743, 47.491, 62.372, -26.835]
  Call Extruder(463.04061)
  MoveL 10291 to (-27.03, 35.64, 144.49) mm, rotated rx 180 ry 0 rz 180 deg; joints [-139.256, -43.507, -98.716, 47.464, 62.347, -26.833]
  MoveL 10292 to (-27.03, 35.64, 144.49) mm, rotated rx 180 ry 0 rz 180 deg; joints [-139.256, -43.507, -98.716, 47.464, 62.347, -26.833]
  Call Extruder(463.20270)
  MoveL 10293 to (-26.72, 35.59, 144.49) mm, rotated rx -180 ry 0 rz 180 deg; joints [-139.294, -43.521, -98.681, 47.433, 62.316, -26.832]
  MoveL 10294 to (-26.72, 35.59, 144.49) mm, rotated rx -180 ry 0 rz 180 deg; joints [-139.294, -43.521, -98.681, 47.433, 62.316, -26.832]
  Call Extruder(463.36408)
  MoveL 10295 to (-26.41, 35.54, 144.49) mm, rotated rx -180 ry 0 rz -180 deg; joints [-139.332, -43.536, -98.646, 47.403, 62.284, -26.831]
  MoveL 10296 to (-26.41, 35.54, 144.49) mm, rotated rx -180 ry 0 rz -180 deg; joints [-139.332, -43.536, -98.646, 47.403, 62.284, -26.831]
  Call Extruder(463.52472)
  MoveL 10297 to (-26.11, 35.49, 144.49) mm, rotated rx 180 ry 0 rz -180 deg; joints [-139.371, -43.55, -98.611, 47.372, 62.253, -26.83]
  MoveL 10298 to (-26.11, 35.49, 144.49) mm, rotated rx 180 ry 0 rz -180 deg; joints [-139.371, -43.55, -98.611, 47.372, 62.253, -26.83]
  Call Extruder(463.68463)
  MoveL 10299 to (-25.8, 35.44, 144.49) mm, rotated rx 180 ry 0 rz 180 deg; joints [-139.409, -43.564, -98.576, 47.342, 62.222, -26.829]
  MoveL 10300 to (-25.8, 35.44, 144.49) mm, rotated rx 180 ry 0 rz 180 deg; joints [-139.409, -43.564, -98.576, 47.342, 62.222, -26.829]
  Call Extruder(463.84382)
  MoveL 10301 to (-25.5, 35.39, 144.49) mm, rotated rx 180 ry 0 rz 180 deg; joints [-139.447, -43.579, -98.541, 47.311, 62.191, -26.829]
  MoveL 10302 to (-25.5, 35.39, 144.49) mm, rotated rx 180 ry 0 rz 180 deg; joints [-139.447, -43.579, -98.541, 47.311, 62.191, -26.829]
  Call Extruder(464.00228)
  MoveL 10303 to (-25.19, 35.34, 144.49) mm, rotated rx -180 ry 0 rz -180 deg; joints [-139.485, -43.593, -98.506, 47.281, 62.16, -26.828]
  MoveL 10304 to (-25.19, 35.34, 144.49) mm, rotated rx -180 ry 0 rz -180 deg; joints [-139.485, -43.593, -98.506, 47.281, 62.16, -26.828]
  Call Extruder(464.20116)
  MoveL 10305 to (-24.8, 35.3, 144.49) mm, rotated rx 180 ry 0 rz 180 deg; joints [-139.531, -43.612, -98.46, 47.244, 62.121, -26.828]
  MoveL 10306 to (-24.8, 35.3, 144.49) mm, rotated rx 180 ry 0 rz 180 deg; joints [-139.531, -43.612, -98.46, 47.244, 62.121, -26.828]
  Call Extruder(464.39916)
  MoveL 10307 to (-24.42, 35.25, 144.49) mm, rotated rx -180 ry 0 rz 180 deg; joints [-139.577, -43.632, -98.414, 47.208, 62.082, -26.829]
  MoveL 10308 to (-24.42, 35.25, 144.49) mm, rotated rx -180 ry 0 rz 180 deg; joints [-139.577, -43.632, -98.414, 47.208, 62.082, -26.829]
  Call Extruder(464.59630)
  MoveL 10309 to (-24.03, 35.21, 144.49) mm, rotated rx -180 ry 0 rz 180 deg; joints [-139.624, -43.651, -98.368, 47.172, 62.042, -26.829]
  MoveL 10310 to (-24.03, 35.21, 144.49) mm, rotated rx -180 ry 0 rz 180 deg; joints [-139.624, -43.651, -98.368, 47.172, 62.042, -26.829]
  Call Extruder(464.79258)
  MoveL 10311 to (-23.64, 35.16, 144.49) mm, rotated rx 180 ry 0 rz 180 deg; joints [-139.67, -43.67, -98.322, 47.136, 62.003, -26.83]
  MoveL 10312 to (-23.64, 35.16, 144.49) mm, rotated rx 180 ry 0 rz 180 deg; joints [-139.67, -43.67, -98.322, 47.136, 62.003, -26.83]
  Call Extruder(465.03826)
  MoveL 10313 to (-23.15, 35.11, 144.49) mm, rotated rx 180 ry 0 rz -180 deg; joints [-139.726, -43.695, -98.262, 47.093, 61.954, -26.832]
  MoveL 10314 to (-23.15, 35.11, 144.49) mm, rotated rx 180 ry 0 rz -180 deg; joints [-139.726, -43.695, -98.262, 47.093, 61.954, -26.832]
  Call Extruder(465.33299)
  MoveL 10315 to (-22.56, 35.07, 144.49) mm, rotated rx 180 ry 0 rz -180 deg; joints [-139.793, -43.725, -98.189, 47.042, 61.894, -26.836]
  MoveL 10316 to (-22.56, 35.07, 144.49) mm, rotated rx 180 ry 0 rz -180 deg; joints [-139.793, -43.725, -98.189, 47.042, 61.894, -26.836]
  Call Extruder(465.62639)
  MoveL 10317 to (-21.97, 35.02, 144.49) mm, rotated rx 180 ry 0 rz 180 deg; joints [-139.86, -43.755, -98.115, 46.991, 61.835, -26.84]
  MoveL 10318 to (-21.97, 35.02, 144.49) mm, rotated rx 180 ry 0 rz 180 deg; joints [-139.86, -43.755, -98.115, 46.991, 61.835, -26.84]
  Call Extruder(466.05972)
  MoveL 10319 to (-21.1, 34.98, 144.49) mm, rotated rx 180 ry 0 rz 180 deg; joints [-139.956, -43.802, -98.004, 46.919, 61.747, -26.848]
  MoveL 10320 to (-21.1, 34.98, 144.49) mm, rotated rx 180 ry 0 rz 180 deg; joints [-139.956, -43.802, -98.004, 46.919, 61.747, -26.848]
  Call Extruder(466.63188)
  MoveL 10321 to (-19.94, 34.93, 144.49) mm, rotated rx 180 ry 0 rz -180 deg; joints [-140.081, -43.865, -97.853, 46.827, 61.63, -26.861]
  MoveL 10322 to (-19.94, 34.93, 144.49) mm, rotated rx 180 ry 0 rz -180 deg; joints [-140.081, -43.865, -97.853, 46.827, 61.63, -26.861]
  Call Extruder(467.05971)
  MoveL 10323 to (-19.06, 34.91, 144.49) mm, rotated rx -180 ry 0 rz 180 deg; joints [-140.173, -43.913, -97.738, 46.76, 61.543, -26.872]
  Call Extruder(583.70842)
  MoveL 10324 to (219.06, 34.91, 144.49) mm, rotated rx 180 ry 0 rz 180 deg; joints [-155.896, -63.38, -55.434, 42.869, 36.89, -36.591]
  MoveL 10325 to (219.06, 34.91, 144.49) mm, rotated rx 180 ry 0 rz 180 deg; joints [-155.896, -63.38, -55.434, 42.869, 36.89, -36.591]
  Call Extruder(584.42399)
  MoveL 10326 to (220.52, 34.95, 144.49) mm, rotated rx 180 ry 0 rz -180 deg; joints [-155.953, -63.552, -55.083, 42.957, 36.725, -36.734]
  MoveL 10327 to (220.52, 34.95, 144.49) mm, rotated rx 180 ry 0 rz -180 deg; joints [-155.953, -63.552, -55.083, 42.957, 36.725, -36.734]
  Call Extruder(584.99873)
  MoveL 10328 to (221.68, 35, 144.49) mm, rotated rx 180 ry 0 rz 180 deg; joints [-155.997, -63.69, -54.8, 43.031, 36.593, -36.852]
  MoveL 10329 to (221.68, 35, 144.49) mm, rotated rx 180 ry 0 rz 180 deg; joints [-155.997, -63.69, -54.8, 43.031, 36.593, -36.852]
  Call Extruder(585.29212)
  MoveL 10330 to (222.27, 35.04, 144.49) mm, rotated rx 180 ry 0 rz 180 deg; joints [-156.017, -63.762, -54.653, 43.073, 36.526, -36.917]
  MoveL 10331 to (222.27, 35.04, 144.49) mm, rotated rx 180 ry 0 rz 180 deg; joints [-156.017, -63.762, -54.653, 43.073, 36.526, -36.917]
  Call Extruder(585.58685)
  MoveL 10332 to (222.86, 35.09, 144.49) mm, rotated rx -180 ry 0 rz -180 deg; joints [-156.037, -63.834, -54.507, 43.115, 36.459, -36.981]
  MoveL 10333 to (222.86, 35.09, 144.49) mm, rotated rx -180 ry 0 rz -180 deg; joints [-156.037, -63.834, -54.507, 43.115, 36.459, -36.981]
  Call Extruder(585.88292)
  MoveL 10334 to (223.45, 35.14, 144.49) mm, rotated rx -180 ry 0 rz 180 deg; joints [-156.057, -63.906, -54.359, 43.158, 36.392, -37.046]
  MoveL 10335 to (223.45, 35.14, 144.49) mm, rotated rx -180 ry 0 rz 180 deg; joints [-156.057, -63.906, -54.359, 43.158, 36.392, -37.046]
  Call Extruder(586.07919)
  MoveL 10336 to (223.83, 35.18, 144.49) mm, rotated rx 180 ry 0 rz -180 deg; joints [-156.068, -63.954, -54.261, 43.189, 36.349, -37.091]
  MoveL 10337 to (223.83, 35.18, 144.49) mm, rotated rx 180 ry 0 rz -180 deg; joints [-156.068, -63.954, -54.261, 43.189, 36.349, -37.091]
  Call Extruder(586.27633)
  MoveL 10338 to (224.22, 35.23, 144.49) mm, rotated rx 180 ry 0 rz 180 deg; joints [-156.08, -64.002, -54.162, 43.22, 36.305, -37.137]
  MoveL 10339 to (224.22, 35.23, 144.49) mm, rotated rx 180 ry 0 rz 180 deg; joints [-156.08, -64.002, -54.162, 43.22, 36.305, -37.137]
  Call Extruder(586.47434)
  MoveL 10340 to (224.61, 35.27, 144.49) mm, rotated rx -180 ry 0 rz 180 deg; joints [-156.092, -64.05, -54.064, 43.252, 36.261, -37.183]
  MoveL 10341 to (224.61, 35.27, 144.49) mm, rotated rx -180 ry 0 rz 180 deg; joints [-156.092, -64.05, -54.064, 43.252, 36.261, -37.183]
  Call Extruder(586.67322)
  MoveL 10342 to (225, 35.32, 144.49) mm, rotated rx 180 ry 0 rz -180 deg; joints [-156.103, -64.099, -53.965, 43.283, 36.217, -37.229]
  MoveL 10343 to (225, 35.32, 144.49) mm, rotated rx 180 ry 0 rz -180 deg; joints [-156.103, -64.099, -53.965, 43.283, 36.217, -37.229]
  Call Extruder(586.85230)
  MoveL 10344 to (225.34, 35.37, 144.49) mm, rotated rx -180 ry 0 rz 180 deg; joints [-156.113, -64.143, -53.876, 43.313, 36.178, -37.271]
  MoveL 10345 to (225.34, 35.37, 144.49) mm, rotated rx -180 ry 0 rz 180 deg; joints [-156.113, -64.143, -53.876, 43.313, 36.178, -37.271]
  Call Extruder(587.01148)
  MoveL 10346 to (225.65, 35.42, 144.49) mm, rotated rx -180 ry 0 rz 180 deg; joints [-156.121, -64.182, -53.796, 43.34, 36.144, -37.309]
  MoveL 10347 to (225.65, 35.42, 144.49) mm, rotated rx -180 ry 0 rz 180 deg; joints [-156.121, -64.182, -53.796, 43.34, 36.144, -37.309]
  Call Extruder(587.17139)
  MoveL 10348 to (225.96, 35.46, 144.49) mm, rotated rx -180 ry 0 rz -180 deg; joints [-156.129, -64.221, -53.716, 43.368, 36.11, -37.348]
  MoveL 10349 to (225.96, 35.46, 144.49) mm, rotated rx -180 ry 0 rz -180 deg; joints [-156.129, -64.221, -53.716, 43.368, 36.11, -37.348]
  Call Extruder(587.33203)
  MoveL 10350 to (226.26, 35.51, 144.49) mm, rotated rx 180 ry 0 rz 180 deg; joints [-156.137, -64.26, -53.637, 43.395, 36.075, -37.387]
  MoveL 10351 to (226.26, 35.51, 144.49) mm, rotated rx 180 ry 0 rz 180 deg; joints [-156.137, -64.26, -53.637, 43.395, 36.075, -37.387]
  Call Extruder(587.49340)
  MoveL 10352 to (226.57, 35.56, 144.49) mm, rotated rx 180 ry 0 rz -180 deg; joints [-156.145, -64.299, -53.557, 43.423, 36.041, -37.426]
  MoveL 10353 to (226.57, 35.56, 144.49) mm, rotated rx 180 ry 0 rz -180 deg; joints [-156.145, -64.299, -53.557, 43.423, 36.041, -37.426]
  Call Extruder(587.65549)
  MoveL 10354 to (226.87, 35.61, 144.49) mm, rotated rx -180 ry 0 rz 180 deg; joints [-156.153, -64.338, -53.477, 43.451, 36.006, -37.465]
  MoveL 10355 to (226.87, 35.61, 144.49) mm, rotated rx -180 ry 0 rz 180 deg; joints [-156.153, -64.338, -53.477, 43.451, 36.006, -37.465]
  Call Extruder(587.80369)
  MoveL 10356 to (227.15, 35.66, 144.49) mm, rotated rx 180 ry 0 rz 180 deg; joints [-156.16, -64.374, -53.404, 43.477, 35.975, -37.501]
  MoveL 10357 to (227.15, 35.66, 144.49) mm, rotated rx 180 ry 0 rz 180 deg; joints [-156.16, -64.374, -53.404, 43.477, 35.975, -37.501]
  Call Extruder(587.93792)
  MoveL 10358 to (227.4, 35.71, 144.49) mm, rotated rx -180 ry 0 rz 180 deg; joints [-156.165, -64.406, -53.337, 43.501, 35.947, -37.534]
  MoveL 10359 to (227.4, 35.71, 144.49) mm, rotated rx -180 ry 0 rz 180 deg; joints [-156.165, -64.406, -53.337, 43.501, 35.947, -37.534]
  Call Extruder(588.07276)
  MoveL 10360 to (227.65, 35.76, 144.49) mm, rotated rx 180 ry 0 rz 180 deg; joints [-156.171, -64.439, -53.271, 43.526, 35.919, -37.568]
  MoveL 10361 to (227.65, 35.76, 144.49) mm, rotated rx 180 ry 0 rz 180 deg; joints [-156.171, -64.439, -53.271, 43.526, 35.919, -37.568]
  Call Extruder(588.20822)
  MoveL 10362 to (227.9, 35.81, 144.49) mm, rotated rx -180 ry 0 rz 180 deg; joints [-156.176, -64.471, -53.205, 43.551, 35.891, -37.602]
  MoveL 10363 to (227.9, 35.81, 144.49) mm, rotated rx -180 ry 0 rz 180 deg; joints [-156.176, -64.471, -53.205, 43.551, 35.891, -37.602]
  Call Extruder(588.34428)
  MoveL 10364 to (228.15, 35.86, 144.49) mm, rotated rx 180 ry 0 rz 180 deg; joints [-156.182, -64.504, -53.138, 43.576, 35.863, -37.635]
  MoveL 10365 to (228.15, 35.86, 144.49) mm, rotated rx 180 ry 0 rz 180 deg; joints [-156.182, -64.504, -53.138, 43.576, 35.863, -37.635]
  Call Extruder(588.48095)
  MoveL 10366 to (228.4, 35.91, 144.49) mm, rotated rx 180 ry 0 rz 180 deg; joints [-156.187, -64.537, -53.071, 43.6, 35.835, -37.669]
  MoveL 10367 to (228.4, 35.91, 144.49) mm, rotated rx 180 ry 0 rz 180 deg; joints [-156.187, -64.537, -53.071, 43.6, 35.835, -37.669]
  Call Extruder(588.61823)
  MoveL 10368 to (228.64, 35.96, 144.49) mm, rotated rx 180 ry 0 rz -180 deg; joints [-156.193, -64.569, -53.005, 43.625, 35.807, -37.703]
  MoveL 10369 to (228.64, 35.96, 144.49) mm, rotated rx 180 ry 0 rz -180 deg; joints [-156.193, -64.569, -53.005, 43.625, 35.807, -37.703]
  Call Extruder(588.74391)
  MoveL 10370 to (228.87, 36, 144.49) mm, rotated rx 180 ry 0 rz 180 deg; joints [-156.198, -64.599, -52.944, 43.649, 35.782, -37.735]
  MoveL 10371 to (228.87, 36, 144.49) mm, rotated rx 180 ry 0 rz 180 deg; joints [-156.198, -64.599, -52.944, 43.649, 35.782, -37.735]
  Call Extruder(588.85785)
  MoveL 10372 to (229.08, 36.05, 144.49) mm, rotated rx -180 ry 0 rz -180 deg; joints [-156.202, -64.626, -52.889, 43.67, 35.759, -37.763]
  MoveL 10373 to (229.08, 36.05, 144.49) mm, rotated rx -180 ry 0 rz -180 deg; joints [-156.202, -64.626, -52.889, 43.67, 35.759, -37.763]
  Call Extruder(588.97225)
  MoveL 10374 to (229.28, 36.09, 144.49) mm, rotated rx 180 ry 0 rz -180 deg; joints [-156.206, -64.653, -52.834, 43.691, 35.736, -37.792]
  MoveL 10375 to (229.28, 36.09, 144.49) mm, rotated rx 180 ry 0 rz -180 deg; joints [-156.206, -64.653, -52.834, 43.691, 35.736, -37.792]
  Call Extruder(589.08710)
  MoveL 10376 to (229.48, 36.14, 144.49) mm, rotated rx 180 ry 0 rz 180 deg; joints [-156.21, -64.68, -52.778, 43.713, 35.713, -37.821]
  MoveL 10377 to (229.48, 36.14, 144.49) mm, rotated rx 180 ry 0 rz 180 deg; joints [-156.21, -64.68, -52.778, 43.713, 35.713, -37.821]
  Call Extruder(589.20240)
  MoveL 10378 to (229.69, 36.18, 144.49) mm, rotated rx 180 ry 0 rz -180 deg; joints [-156.214, -64.708, -52.723, 43.734, 35.691, -37.849]
  MoveL 10379 to (229.69, 36.18, 144.49) mm, rotated rx 180 ry 0 rz -180 deg; joints [-156.214, -64.708, -52.723, 43.734, 35.691, -37.849]
  Call Extruder(589.26695)
  MoveL 10380 to (229.8, 36.22, 144.49) mm, rotated rx 180 ry 0 rz 180 deg; joints [-156.216, -64.723, -52.692, 43.747, 35.678, -37.867]
  MoveL 10381 to (229.8, 36.22, 144.49) mm, rotated rx 180 ry 0 rz 180 deg; joints [-156.216, -64.723, -52.692, 43.747, 35.678, -37.867]
  Call Extruder(589.39662)
  MoveL 10382 to (230.02, 36.28, 144.49) mm, rotated rx 180 ry 0 rz -180 deg; joints [-156.219, -64.754, -52.629, 43.774, 35.653, -37.901]
  MoveL 10383 to (230.02, 36.28, 144.49) mm, rotated rx 180 ry 0 rz -180 deg; joints [-156.219, -64.754, -52.629, 43.774, 35.653, -37.901]
  Call Extruder(589.52685)
  MoveL 10384 to (230.25, 36.35, 144.49) mm, rotated rx -180 ry 0 rz 180 deg; joints [-156.221, -64.784, -52.566, 43.801, 35.629, -37.936]
  MoveL 10385 to (230.25, 36.35, 144.49) mm, rotated rx -180 ry 0 rz 180 deg; joints [-156.221, -64.784, -52.566, 43.801, 35.629, -37.936]
  Call Extruder(589.65764)
  MoveL 10386 to (230.47, 36.42, 144.49) mm, rotated rx 180 ry 0 rz -180 deg; joints [-156.224, -64.815, -52.504, 43.828, 35.604, -37.971]
  MoveL 10387 to (230.47, 36.42, 144.49) mm, rotated rx 180 ry 0 rz -180 deg; joints [-156.224, -64.815, -52.504, 43.828, 35.604, -37.971]
  Call Extruder(589.78900)
  MoveL 10388 to (230.69, 36.49, 144.49) mm, rotated rx 180 ry 0 rz 180 deg; joints [-156.227, -64.846, -52.441, 43.856, 35.579, -38.006]
  MoveL 10389 to (230.69, 36.49, 144.49) mm, rotated rx 180 ry 0 rz 180 deg; joints [-156.227, -64.846, -52.441, 43.856, 35.579, -38.006]
  Call Extruder(589.90090)
  MoveL 10390 to (230.88, 36.55, 144.49) mm, rotated rx 180 ry 0 rz 180 deg; joints [-156.229, -64.872, -52.387, 43.879, 35.558, -38.036]
  MoveL 10391 to (230.88, 36.55, 144.49) mm, rotated rx 180 ry 0 rz 180 deg; joints [-156.229, -64.872, -52.387, 43.879, 35.558, -38.036]
  Call Extruder(590.01324)
  MoveL 10392 to (231.07, 36.61, 144.49) mm, rotated rx 180 ry 0 rz 180 deg; joints [-156.231, -64.899, -52.334, 43.903, 35.537, -38.067]
  MoveL 10393 to (231.07, 36.61, 144.49) mm, rotated rx 180 ry 0 rz 180 deg; joints [-156.231, -64.899, -52.334, 43.903, 35.537, -38.067]
  Call Extruder(590.12603)
  MoveL 10394 to (231.26, 36.67, 144.49) mm, rotated rx 180 ry 0 rz 180 deg; joints [-156.233, -64.925, -52.28, 43.927, 35.516, -38.097]
  MoveL 10395 to (231.26, 36.67, 144.49) mm, rotated rx 180 ry 0 rz 180 deg; joints [-156.233, -64.925, -52.28, 43.927, 35.516, -38.097]
  Call Extruder(590.23926)
  MoveL 10396 to (231.45, 36.73, 144.49) mm, rotated rx 180 ry 0 rz 180 deg; joints [-156.235, -64.951, -52.226, 43.951, 35.495, -38.127]
  MoveL 10397 to (231.45, 36.73, 144.49) mm, rotated rx 180 ry 0 rz 180 deg; joints [-156.235, -64.951, -52.226, 43.951, 35.495, -38.127]
  Call Extruder(590.35294)
  MoveL 10398 to (231.64, 36.79, 144.49) mm, rotated rx -180 ry 0 rz 180 deg; joints [-156.237, -64.978, -52.173, 43.974, 35.475, -38.158]
  MoveL 10399 to (231.64, 36.79, 144.49) mm, rotated rx -180 ry 0 rz 180 deg; joints [-156.237, -64.978, -52.173, 43.974, 35.475, -38.158]
  Call Extruder(590.53490)
  MoveL 10400 to (231.93, 36.91, 144.49) mm, rotated rx -180 ry 0 rz 180 deg; joints [-156.238, -65.02, -52.087, 44.016, 35.443, -38.209]
  MoveL 10401 to (231.93, 36.91, 144.49) mm, rotated rx -180 ry 0 rz 180 deg; joints [-156.238, -65.02, -52.087, 44.016, 35.443, -38.209]
  Call Extruder(590.71761)
  MoveL 10402 to (232.22, 37.03, 144.49) mm, rotated rx 180 ry 0 rz 180 deg; joints [-156.238, -65.062, -52.001, 44.058, 35.411, -38.261]
  MoveL 10403 to (232.22, 37.03, 144.49) mm, rotated rx 180 ry 0 rz 180 deg; joints [-156.238, -65.062, -52.001, 44.058, 35.411, -38.261]
  Call Extruder(590.88803)
  MoveL 10404 to (232.49, 37.15, 144.49) mm, rotated rx -180 ry 0 rz 180 deg; joints [-156.239, -65.101, -51.921, 44.097, 35.381, -38.31]
  MoveL 10405 to (232.49, 37.15, 144.49) mm, rotated rx -180 ry 0 rz 180 deg; joints [-156.239, -65.101, -51.921, 44.097, 35.381, -38.31]
  Call Extruder(591.04603)
  MoveL 10406 to (232.74, 37.26, 144.49) mm, rotated rx 180 ry 0 rz 180 deg; joints [-156.239, -65.138, -51.847, 44.134, 35.354, -38.355]
  MoveL 10407 to (232.74, 37.26, 144.49) mm, rotated rx 180 ry 0 rz 180 deg; joints [-156.239, -65.138, -51.847, 44.134, 35.354, -38.355]
  Call Extruder(591.20464)
  MoveL 10408 to (232.99, 37.36, 144.49) mm, rotated rx 180 ry 0 rz -180 deg; joints [-156.239, -65.174, -51.773, 44.171, 35.327, -38.4]
  MoveL 10409 to (232.99, 37.36, 144.49) mm, rotated rx 180 ry 0 rz -180 deg; joints [-156.239, -65.174, -51.773, 44.171, 35.327, -38.4]
  Call Extruder(591.41080)
  MoveL 10410 to (233.29, 37.54, 144.49) mm, rotated rx -180 ry 0 rz 180 deg; joints [-156.236, -65.221, -51.677, 44.224, 35.294, -38.462]
  MoveL 10411 to (233.29, 37.54, 144.49) mm, rotated rx -180 ry 0 rz 180 deg; joints [-156.236, -65.221, -51.677, 44.224, 35.294, -38.462]
  Call Extruder(591.61775)
  MoveL 10412 to (233.6, 37.71, 144.49) mm, rotated rx -180 ry 0 rz -180 deg; joints [-156.232, -65.268, -51.581, 44.277, 35.262, -38.525]
  MoveL 10413 to (233.6, 37.71, 144.49) mm, rotated rx -180 ry 0 rz -180 deg; joints [-156.232, -65.268, -51.581, 44.277, 35.262, -38.525]
  Call Extruder(591.82547)
  MoveL 10414 to (233.9, 37.89, 144.49) mm, rotated rx 180 ry 0 rz 180 deg; joints [-156.228, -65.315, -51.486, 44.33, 35.229, -38.588]
  MoveL 10415 to (233.9, 37.89, 144.49) mm, rotated rx 180 ry 0 rz 180 deg; joints [-156.228, -65.315, -51.486, 44.33, 35.229, -38.588]
  Call Extruder(592.03398)
  MoveL 10416 to (234.21, 38.06, 144.49) mm, rotated rx -180 ry 0 rz 180 deg; joints [-156.224, -65.363, -51.39, 44.383, 35.197, -38.652]
  MoveL 10417 to (234.21, 38.06, 144.49) mm, rotated rx -180 ry 0 rz 180 deg; joints [-156.224, -65.363, -51.39, 44.383, 35.197, -38.652]
  Call Extruder(592.21352)
  MoveL 10418 to (234.45, 38.24, 144.49) mm, rotated rx -180 ry 0 rz 180 deg; joints [-156.218, -65.403, -51.308, 44.433, 35.171, -38.709]
  MoveL 10419 to (234.45, 38.24, 144.49) mm, rotated rx -180 ry 0 rz 180 deg; joints [-156.218, -65.403, -51.308, 44.433, 35.171, -38.709]
  Call Extruder(592.54693)
  MoveL 10420 to (234.9, 38.57, 144.49) mm, rotated rx 180 ry 0 rz 180 deg; joints [-156.206, -65.476, -51.158, 44.524, 35.124, -38.815]
  MoveL 10421 to (234.9, 38.57, 144.49) mm, rotated rx 180 ry 0 rz 180 deg; joints [-156.206, -65.476, -51.158, 44.524, 35.124, -38.815]
  Call Extruder(592.88153)
  MoveL 10422 to (235.35, 38.9, 144.49) mm, rotated rx 180 ry 0 rz -180 deg; joints [-156.195, -65.551, -51.007, 44.617, 35.077, -38.921]
  Call Extruder(593.70948)
  MoveL 10423 to (236.39, 39.81, 144.49) mm, rotated rx 180 ry 0 rz 180 deg; joints [-156.154, -65.73, -50.642, 44.858, 34.971, -39.194]
  Call Extruder(594.53743)
  MoveL 10424 to (237.3, 40.85, 144.49) mm, rotated rx 180 ry 0 rz 180 deg; joints [-156.097, -65.903, -50.293, 45.115, 34.882, -39.476]
  Call Extruder(594.70473)
  MoveL 10425 to (237.47, 41.07, 144.49) mm, rotated rx -180 ry 0 rz 180 deg; joints [-156.083, -65.936, -50.225, 45.168, 34.867, -39.534]
  MoveL 10426 to (237.47, 41.07, 144.49) mm, rotated rx -180 ry 0 rz 180 deg; joints [-156.083, -65.936, -50.225, 45.168, 34.867, -39.534]
  Call Extruder(595.03814)
  MoveL 10427 to (237.8, 41.52, 144.49) mm, rotated rx -180 ry 0 rz 180 deg; joints [-156.055, -66.002, -50.09, 45.275, 34.836, -39.649]
  MoveL 10428 to (237.8, 41.52, 144.49) mm, rotated rx -180 ry 0 rz 180 deg; joints [-156.055, -66.002, -50.09, 45.275, 34.836, -39.649]
  Call Extruder(595.37037)
  MoveL 10429 to (238.12, 41.98, 144.49) mm, rotated rx -180 ry 0 rz -180 deg; joints [-156.028, -66.069, -49.954, 45.383, 34.805, -39.765]
  MoveL 10430 to (238.12, 41.98, 144.49) mm, rotated rx -180 ry 0 rz -180 deg; joints [-156.028, -66.069, -49.954, 45.383, 34.805, -39.765]
  Call Extruder(595.48807)
  MoveL 10431 to (238.22, 42.15, 144.49) mm, rotated rx 180 ry 0 rz 180 deg; joints [-156.016, -66.092, -49.91, 45.421, 34.796, -39.806]
  MoveL 10432 to (238.22, 42.15, 144.49) mm, rotated rx 180 ry 0 rz 180 deg; joints [-156.016, -66.092, -49.91, 45.421, 34.796, -39.806]
  Call Extruder(595.69580)
  MoveL 10433 to (238.4, 42.45, 144.49) mm, rotated rx 180 ry 0 rz 180 deg; joints [-155.996, -66.131, -49.83, 45.49, 34.781, -39.879]
  MoveL 10434 to (238.4, 42.45, 144.49) mm, rotated rx 180 ry 0 rz 180 deg; joints [-155.996, -66.131, -49.83, 45.49, 34.781, -39.879]
  Call Extruder(595.90274)
  MoveL 10435 to (238.57, 42.75, 144.49) mm, rotated rx 180 ry 0 rz -180 deg; joints [-155.976, -66.17, -49.75, 45.559, 34.765, -39.952]
  MoveL 10436 to (238.57, 42.75, 144.49) mm, rotated rx 180 ry 0 rz -180 deg; joints [-155.976, -66.17, -49.75, 45.559, 34.765, -39.952]
  Call Extruder(596.10891)
  MoveL 10437 to (238.75, 43.06, 144.49) mm, rotated rx 180 ry 0 rz 180 deg; joints [-155.956, -66.21, -49.67, 45.628, 34.75, -40.025]
  MoveL 10438 to (238.75, 43.06, 144.49) mm, rotated rx 180 ry 0 rz 180 deg; joints [-155.956, -66.21, -49.67, 45.628, 34.75, -40.025]
  Call Extruder(596.29060)
  MoveL 10439 to (238.89, 43.33, 144.49) mm, rotated rx -180 ry 0 rz 180 deg; joints [-155.937, -66.244, -49.601, 45.689, 34.738, -40.09]
  MoveL 10440 to (238.89, 43.33, 144.49) mm, rotated rx -180 ry 0 rz 180 deg; joints [-155.937, -66.244, -49.601, 45.689, 34.738, -40.09]
  Call Extruder(596.44861)
  MoveL 10441 to (239, 43.58, 144.49) mm, rotated rx -180 ry 0 rz -180 deg; joints [-155.919, -66.271, -49.545, 45.743, 34.73, -40.146]
  MoveL 10442 to (239, 43.58, 144.49) mm, rotated rx -180 ry 0 rz -180 deg; joints [-155.919, -66.271, -49.545, 45.743, 34.73, -40.146]
  Call Extruder(596.60601)
  MoveL 10443 to (239.1, 43.83, 144.49) mm, rotated rx 180 ry 0 rz -180 deg; joints [-155.901, -66.299, -49.489, 45.797, 34.722, -40.202]
  MoveL 10444 to (239.1, 43.83, 144.49) mm, rotated rx 180 ry 0 rz -180 deg; joints [-155.901, -66.299, -49.489, 45.797, 34.722, -40.202]
  Call Extruder(596.78872)
  MoveL 10445 to (239.23, 44.12, 144.49) mm, rotated rx 180 ry 0 rz 180 deg; joints [-155.879, -66.331, -49.424, 45.859, 34.713, -40.266]
  MoveL 10446 to (239.23, 44.12, 144.49) mm, rotated rx 180 ry 0 rz 180 deg; joints [-155.879, -66.331, -49.424, 45.859, 34.713, -40.266]
  Call Extruder(596.97068)
  MoveL 10447 to (239.35, 44.42, 144.49) mm, rotated rx 180 ry 0 rz -180 deg; joints [-155.858, -66.363, -49.359, 45.922, 34.703, -40.331]
  MoveL 10448 to (239.35, 44.42, 144.49) mm, rotated rx 180 ry 0 rz -180 deg; joints [-155.858, -66.363, -49.359, 45.922, 34.703, -40.331]
  Call Extruder(597.11801)
  MoveL 10449 to (239.44, 44.66, 144.49) mm, rotated rx 180 ry 0 rz -180 deg; joints [-155.84, -66.388, -49.308, 45.973, 34.697, -40.384]
  MoveL 10450 to (239.44, 44.66, 144.49) mm, rotated rx 180 ry 0 rz -180 deg; joints [-155.84, -66.388, -49.308, 45.973, 34.697, -40.384]
  Call Extruder(597.23124)
  MoveL 10451 to (239.5, 44.85, 144.49) mm, rotated rx 180 ry 0 rz 180 deg; joints [-155.826, -66.407, -49.27, 46.012, 34.693, -40.424]
  MoveL 10452 to (239.5, 44.85, 144.49) mm, rotated rx 180 ry 0 rz 180 deg; joints [-155.826, -66.407, -49.27, 46.012, 34.693, -40.424]
  Call Extruder(597.34404)
  MoveL 10453 to (239.56, 45.03, 144.49) mm, rotated rx -180 ry 0 rz -180 deg; joints [-155.811, -66.426, -49.232, 46.051, 34.689, -40.464]
  MoveL 10454 to (239.56, 45.03, 144.49) mm, rotated rx -180 ry 0 rz -180 deg; joints [-155.811, -66.426, -49.232, 46.051, 34.689, -40.464]
  Call Extruder(597.45638)
  MoveL 10455 to (239.62, 45.22, 144.49) mm, rotated rx 180 ry 0 rz -180 deg; joints [-155.797, -66.444, -49.194, 46.09, 34.685, -40.504]
  MoveL 10456 to (239.62, 45.22, 144.49) mm, rotated rx 180 ry 0 rz -180 deg; joints [-155.797, -66.444, -49.194, 46.09, 34.685, -40.504]
  Call Extruder(597.56829)
  MoveL 10457 to (239.68, 45.41, 144.49) mm, rotated rx 180 ry 0 rz 180 deg; joints [-155.783, -66.463, -49.157, 46.129, 34.681, -40.544]
  MoveL 10458 to (239.68, 45.41, 144.49) mm, rotated rx 180 ry 0 rz 180 deg; joints [-155.783, -66.463, -49.157, 46.129, 34.681, -40.544]
  Call Extruder(597.68969)
  MoveL 10459 to (239.75, 45.62, 144.49) mm, rotated rx 180 ry 0 rz 180 deg; joints [-155.767, -66.483, -49.116, 46.172, 34.677, -40.587]
  MoveL 10460 to (239.75, 45.62, 144.49) mm, rotated rx 180 ry 0 rz 180 deg; joints [-155.767, -66.483, -49.116, 46.172, 34.677, -40.587]
  Call Extruder(597.82048)
  MoveL 10461 to (239.81, 45.84, 144.49) mm, rotated rx -180 ry 0 rz 180 deg; joints [-155.75, -66.505, -49.072, 46.218, 34.673, -40.634]
  MoveL 10462 to (239.81, 45.84, 144.49) mm, rotated rx -180 ry 0 rz 180 deg; joints [-155.75, -66.505, -49.072, 46.218, 34.673, -40.634]
  Call Extruder(597.95070)
  MoveL 10463 to (239.88, 46.06, 144.49) mm, rotated rx 180 ry 0 rz 180 deg; joints [-155.733, -66.526, -49.029, 46.264, 34.669, -40.681]
  MoveL 10464 to (239.88, 46.06, 144.49) mm, rotated rx 180 ry 0 rz 180 deg; joints [-155.733, -66.526, -49.029, 46.264, 34.669, -40.681]
  Call Extruder(598.08036)
  MoveL 10465 to (239.95, 46.29, 144.49) mm, rotated rx 180 ry 0 rz 180 deg; joints [-155.715, -66.548, -48.985, 46.31, 34.665, -40.728]
  MoveL 10466 to (239.95, 46.29, 144.49) mm, rotated rx 180 ry 0 rz 180 deg; joints [-155.715, -66.548, -48.985, 46.31, 34.665, -40.728]
  Call Extruder(598.20946)
  MoveL 10467 to (240.02, 46.51, 144.49) mm, rotated rx -180 ry 0 rz 180 deg; joints [-155.698, -66.569, -48.941, 46.356, 34.661, -40.775]
  MoveL 10468 to (240.02, 46.51, 144.49) mm, rotated rx -180 ry 0 rz 180 deg; joints [-155.698, -66.569, -48.941, 46.356, 34.661, -40.775]
  Call Extruder(598.32451)
  MoveL 10469 to (240.06, 46.72, 144.49) mm, rotated rx 180 ry 0 rz -180 deg; joints [-155.682, -66.587, -48.905, 46.396, 34.659, -40.816]
  MoveL 10470 to (240.06, 46.72, 144.49) mm, rotated rx 180 ry 0 rz -180 deg; joints [-155.682, -66.587, -48.905, 46.396, 34.659, -40.816]
  Call Extruder(598.43912)
  MoveL 10471 to (240.11, 46.92, 144.49) mm, rotated rx -180 ry 0 rz 180 deg; joints [-155.665, -66.605, -48.87, 46.437, 34.657, -40.857]
  MoveL 10472 to (240.11, 46.92, 144.49) mm, rotated rx -180 ry 0 rz 180 deg; joints [-155.665, -66.605, -48.87, 46.437, 34.657, -40.857]
  Call Extruder(598.55327)
  MoveL 10473 to (240.15, 47.12, 144.49) mm, rotated rx 180 ry 0 rz 180 deg; joints [-155.649, -66.622, -48.834, 46.478, 34.656, -40.897]
  MoveL 10474 to (240.15, 47.12, 144.49) mm, rotated rx 180 ry 0 rz 180 deg; joints [-155.649, -66.622, -48.834, 46.478, 34.656, -40.897]
  Call Extruder(598.66696)
  MoveL 10475 to (240.2, 47.33, 144.49) mm, rotated rx 180 ry 0 rz 180 deg; joints [-155.633, -66.64, -48.799, 46.519, 34.654, -40.939]
  MoveL 10476 to (240.2, 47.33, 144.49) mm, rotated rx 180 ry 0 rz 180 deg; joints [-155.633, -66.64, -48.799, 46.519, 34.654, -40.939]
  Call Extruder(598.79237)
  MoveL 10477 to (240.24, 47.55, 144.49) mm, rotated rx 180 ry 0 rz 180 deg; joints [-155.614, -66.659, -48.76, 46.563, 34.652, -40.984]
  MoveL 10478 to (240.24, 47.55, 144.49) mm, rotated rx 180 ry 0 rz 180 deg; joints [-155.614, -66.659, -48.76, 46.563, 34.652, -40.984]
  Call Extruder(598.92935)
  MoveL 10479 to (240.29, 47.8, 144.49) mm, rotated rx 180 ry 0 rz 180 deg; joints [-155.594, -66.68, -48.717, 46.613, 34.651, -41.033]
  MoveL 10480 to (240.29, 47.8, 144.49) mm, rotated rx 180 ry 0 rz 180 deg; joints [-155.594, -66.68, -48.717, 46.613, 34.651, -41.033]
  Call Extruder(599.06572)
  MoveL 10481 to (240.34, 48.05, 144.49) mm, rotated rx 180 ry 0 rz 180 deg; joints [-155.574, -66.701, -48.675, 46.662, 34.649, -41.082]
  MoveL 10482 to (240.34, 48.05, 144.49) mm, rotated rx 180 ry 0 rz 180 deg; joints [-155.574, -66.701, -48.675, 46.662, 34.649, -41.082]
  Call Extruder(599.20147)
  MoveL 10483 to (240.39, 48.3, 144.49) mm, rotated rx 180 ry 0 rz 180 deg; joints [-155.554, -66.722, -48.632, 46.711, 34.648, -41.132]
  MoveL 10484 to (240.39, 48.3, 144.49) mm, rotated rx 180 ry 0 rz 180 deg; joints [-155.554, -66.722, -48.632, 46.711, 34.648, -41.132]
  Call Extruder(599.33662)
  MoveL 10485 to (240.44, 48.55, 144.49) mm, rotated rx -180 ry 0 rz 180 deg; joints [-155.534, -66.743, -48.59, 46.76, 34.646, -41.181]
  MoveL 10486 to (240.44, 48.55, 144.49) mm, rotated rx -180 ry 0 rz 180 deg; joints [-155.534, -66.743, -48.59, 46.76, 34.646, -41.181]
  Call Extruder(599.47116)
  MoveL 10487 to (240.49, 48.8, 144.49) mm, rotated rx -180 ry 0 rz 180 deg; joints [-155.514, -66.764, -48.548, 46.81, 34.645, -41.231]
  MoveL 10488 to (240.49, 48.8, 144.49) mm, rotated rx -180 ry 0 rz 180 deg; joints [-155.514, -66.764, -48.548, 46.81, 34.645, -41.231]
  Call Extruder(599.60508)
  MoveL 10489 to (240.54, 49.05, 144.49) mm, rotated rx 180 ry 0 rz 180 deg; joints [-155.494, -66.785, -48.505, 46.859, 34.643, -41.28]
  MoveL 10490 to (240.54, 49.05, 144.49) mm, rotated rx 180 ry 0 rz 180 deg; joints [-155.494, -66.785, -48.505, 46.859, 34.643, -41.28]
  Call Extruder(599.75295)
  MoveL 10491 to (240.59, 49.33, 144.49) mm, rotated rx 180 ry 0 rz -180 deg; joints [-155.471, -66.807, -48.459, 46.913, 34.642, -41.334]
  MoveL 10492 to (240.59, 49.33, 144.49) mm, rotated rx 180 ry 0 rz -180 deg; joints [-155.471, -66.807, -48.459, 46.913, 34.642, -41.334]
  Call Extruder(599.91470)
  MoveL 10493 to (240.64, 49.63, 144.49) mm, rotated rx 180 ry 0 rz -180 deg; joints [-155.446, -66.832, -48.41, 46.973, 34.642, -41.394]
  MoveL 10494 to (240.64, 49.63, 144.49) mm, rotated rx 180 ry 0 rz -180 deg; joints [-155.446, -66.832, -48.41, 46.973, 34.642, -41.394]
  Call Extruder(600.07571)
  MoveL 10495 to (240.69, 49.94, 144.49) mm, rotated rx 180 ry 0 rz 180 deg; joints [-155.421, -66.856, -48.361, 47.032, 34.642, -41.453]
  MoveL 10496 to (240.69, 49.94, 144.49) mm, rotated rx 180 ry 0 rz 180 deg; joints [-155.421, -66.856, -48.361, 47.032, 34.642, -41.453]
  Call Extruder(600.23600)
  MoveL 10497 to (240.74, 50.24, 144.49) mm, rotated rx 180 ry 0 rz 180 deg; joints [-155.396, -66.88, -48.312, 47.092, 34.641, -41.512]
  MoveL 10498 to (240.74, 50.24, 144.49) mm, rotated rx 180 ry 0 rz 180 deg; joints [-155.396, -66.88, -48.312, 47.092, 34.641, -41.512]
  Call Extruder(600.39556)
  MoveL 10499 to (240.78, 50.55, 144.49) mm, rotated rx -180 ry 0 rz 180 deg; joints [-155.371, -66.905, -48.262, 47.151, 34.641, -41.571]
  MoveL 10500 to (240.78, 50.55, 144.49) mm, rotated rx -180 ry 0 rz 180 deg; joints [-155.371, -66.905, -48.262, 47.151, 34.641, -41.571]
  Call Extruder(600.55440)
  MoveL 10501 to (240.83, 50.86, 144.49) mm, rotated rx 180 ry 0 rz -180 deg; joints [-155.346, -66.929, -48.213, 47.211, 34.641, -41.631]
  MoveL 10502 to (240.83, 50.86, 144.49) mm, rotated rx 180 ry 0 rz -180 deg; joints [-155.346, -66.929, -48.213, 47.211, 34.641, -41.631]
  Call Extruder(600.73307)
  MoveL 10503 to (240.88, 51.2, 144.49) mm, rotated rx 180 ry 0 rz -180 deg; joints [-155.317, -66.956, -48.159, 47.277, 34.641, -41.697]
  MoveL 10504 to (240.88, 51.2, 144.49) mm, rotated rx 180 ry 0 rz -180 deg; joints [-155.317, -66.956, -48.159, 47.277, 34.641, -41.697]
  Call Extruder(600.93151)
  MoveL 10505 to (240.93, 51.59, 144.49) mm, rotated rx -180 ry 0 rz -180 deg; joints [-155.285, -66.985, -48.1, 47.351, 34.643, -41.77]
  MoveL 10506 to (240.93, 51.59, 144.49) mm, rotated rx -180 ry 0 rz -180 deg; joints [-155.285, -66.985, -48.1, 47.351, 34.643, -41.77]
  Call Extruder(601.12909)
  MoveL 10507 to (240.97, 51.98, 144.49) mm, rotated rx -180 ry 0 rz 180 deg; joints [-155.252, -67.014, -48.041, 47.425, 34.644, -41.844]
  MoveL 10508 to (240.97, 51.98, 144.49) mm, rotated rx -180 ry 0 rz 180 deg; joints [-155.252, -67.014, -48.041, 47.425, 34.644, -41.844]
  Call Extruder(601.32579)
  MoveL 10509 to (241.02, 52.36, 144.49) mm, rotated rx 180 ry 0 rz 180 deg; joints [-155.22, -67.043, -47.982, 47.5, 34.645, -41.917]
  MoveL 10510 to (241.02, 52.36, 144.49) mm, rotated rx 180 ry 0 rz 180 deg; joints [-155.22, -67.043, -47.982, 47.5, 34.645, -41.917]
  Call Extruder(601.52163)
  MoveL 10511 to (241.06, 52.75, 144.49) mm, rotated rx 180 ry 0 rz 180 deg; joints [-155.188, -67.072, -47.924, 47.573, 34.647, -41.99]
  MoveL 10512 to (241.06, 52.75, 144.49) mm, rotated rx 180 ry 0 rz 180 deg; joints [-155.188, -67.072, -47.924, 47.573, 34.647, -41.99]
  Call Extruder(601.81707)
  MoveL 10513 to (241.11, 53.34, 144.49) mm, rotated rx -180 ry 0 rz 180 deg; joints [-155.138, -67.114, -47.84, 47.684, 34.652, -42.099]
  MoveL 10514 to (241.11, 53.34, 144.49) mm, rotated rx -180 ry 0 rz 180 deg; joints [-155.138, -67.114, -47.84, 47.684, 34.652, -42.099]
  Call Extruder(602.11118)
  MoveL 10515 to (241.16, 53.93, 144.49) mm, rotated rx -180 ry 0 rz 180 deg; joints [-155.088, -67.155, -47.756, 47.795, 34.657, -42.208]
  MoveL 10516 to (241.16, 53.93, 144.49) mm, rotated rx -180 ry 0 rz 180 deg; joints [-155.088, -67.155, -47.756, 47.795, 34.657, -42.208]
  Call Extruder(602.40395)
  MoveL 10517 to (241.2, 54.52, 144.49) mm, rotated rx 180 ry 0 rz 180 deg; joints [-155.038, -67.197, -47.671, 47.906, 34.662, -42.317]
  MoveL 10518 to (241.2, 54.52, 144.49) mm, rotated rx 180 ry 0 rz 180 deg; joints [-155.038, -67.197, -47.671, 47.906, 34.662, -42.317]
  Call Extruder(602.97740)
  MoveL 10519 to (241.25, 55.68, 144.49) mm, rotated rx 180 ry 0 rz 180 deg; joints [-154.938, -67.274, -47.516, 48.12, 34.677, -42.527]
  MoveL 10520 to (241.25, 55.68, 144.49) mm, rotated rx 180 ry 0 rz 180 deg; joints [-154.938, -67.274, -47.516, 48.12, 34.677, -42.527]
  Call Extruder(603.69124)
  MoveL 10521 to (241.29, 57.14, 144.49) mm, rotated rx 180 ry 0 rz 180 deg; joints [-154.812, -67.368, -47.326, 48.386, 34.698, -42.786]
  Call Extruder(645.75613)
  MoveL 10522 to (241.29, 142.86, 144.49) mm, rotated rx -180 ry 0 rz 180 deg; joints [-147.778, -74.094, -33.874, 63.921, 36.416, -58.692]
  Call Extruder(646.18456)
  MoveL 10523 to (241.27, 143.73, 144.49) mm, rotated rx 180 ry 0 rz 180 deg; joints [-147.711, -74.178, -33.707, 64.081, 36.437, -58.865]
  MoveL 10524 to (241.27, 143.73, 144.49) mm, rotated rx 180 ry 0 rz 180 deg; joints [-147.711, -74.178, -33.707, 64.081, 36.437, -58.865]
  Call Extruder(646.75801)
  MoveL 10525 to (241.22, 144.9, 144.49) mm, rotated rx 180 ry 0 rz 180 deg; joints [-147.62, -74.288, -33.489, 64.291, 36.468, -59.091]
  MoveL 10526 to (241.22, 144.9, 144.49) mm, rotated rx 180 ry 0 rz 180 deg; joints [-147.62, -74.288, -33.489, 64.291, 36.468, -59.091]
  Call Extruder(647.19234)
  MoveL 10527 to (241.18, 145.77, 144.49) mm, rotated rx 180 ry 0 rz 180 deg; joints [-147.551, -74.369, -33.328, 64.447, 36.493, -59.26]
  MoveL 10528 to (241.18, 145.77, 144.49) mm, rotated rx 180 ry 0 rz 180 deg; joints [-147.551, -74.369, -33.328, 64.447, 36.493, -59.26]
  Call Extruder(647.48645)
  MoveL 10529 to (241.13, 146.36, 144.49) mm, rotated rx 180 ry 0 rz -180 deg; joints [-147.504, -74.422, -33.225, 64.55, 36.511, -59.37]
  MoveL 10530 to (241.13, 146.36, 144.49) mm, rotated rx 180 ry 0 rz -180 deg; joints [-147.504, -74.422, -33.225, 64.55, 36.511, -59.37]
  Call Extruder(647.78189)
  MoveL 10531 to (241.09, 146.95, 144.49) mm, rotated rx -180 ry 0 rz 180 deg; joints [-147.457, -74.474, -33.12, 64.654, 36.53, -59.481]
  MoveL 10532 to (241.09, 146.95, 144.49) mm, rotated rx -180 ry 0 rz 180 deg; joints [-147.457, -74.474, -33.12, 64.654, 36.53, -59.481]
  Call Extruder(648.02815)
  MoveL 10533 to (241.04, 147.44, 144.49) mm, rotated rx 180 ry 0 rz -180 deg; joints [-147.417, -74.517, -33.036, 64.738, 36.546, -59.571]
  MoveL 10534 to (241.04, 147.44, 144.49) mm, rotated rx 180 ry 0 rz -180 deg; joints [-147.417, -74.517, -33.036, 64.738, 36.546, -59.571]
  Call Extruder(648.22485)
  MoveL 10535 to (240.99, 147.83, 144.49) mm, rotated rx 180 ry 0 rz 180 deg; joints [-147.386, -74.549, -32.972, 64.804, 36.559, -59.641]
  MoveL 10536 to (240.99, 147.83, 144.49) mm, rotated rx 180 ry 0 rz 180 deg; joints [-147.386, -74.549, -32.972, 64.804, 36.559, -59.641]
  Call Extruder(648.42243)
  MoveL 10537 to (240.95, 148.22, 144.49) mm, rotated rx -180 ry 0 rz 180 deg; joints [-147.354, -74.582, -32.907, 64.869, 36.573, -59.711]
  MoveL 10538 to (240.95, 148.22, 144.49) mm, rotated rx -180 ry 0 rz 180 deg; joints [-147.354, -74.582, -32.907, 64.869, 36.573, -59.711]
  Call Extruder(648.62087)
  MoveL 10539 to (240.9, 148.6, 144.49) mm, rotated rx -180 ry 0 rz -180 deg; joints [-147.322, -74.614, -32.843, 64.935, 36.587, -59.781]
  MoveL 10540 to (240.9, 148.6, 144.49) mm, rotated rx -180 ry 0 rz -180 deg; joints [-147.322, -74.614, -32.843, 64.935, 36.587, -59.781]
  Call Extruder(648.82018)
  MoveL 10541 to (240.86, 148.99, 144.49) mm, rotated rx 180 ry 0 rz 180 deg; joints [-147.291, -74.647, -32.779, 65.001, 36.601, -59.851]
  MoveL 10542 to (240.86, 148.99, 144.49) mm, rotated rx 180 ry 0 rz 180 deg; joints [-147.291, -74.647, -32.779, 65.001, 36.601, -59.851]
  Call Extruder(648.97901)
  MoveL 10543 to (240.81, 149.3, 144.49) mm, rotated rx 180 ry 0 rz 180 deg; joints [-147.265, -74.671, -32.731, 65.051, 36.613, -59.904]
  MoveL 10544 to (240.81, 149.3, 144.49) mm, rotated rx 180 ry 0 rz 180 deg; joints [-147.265, -74.671, -32.731, 65.051, 36.613, -59.904]
  Call Extruder(649.13857)
  MoveL 10545 to (240.76, 149.6, 144.49) mm, rotated rx 180 ry 0 rz 180 deg; joints [-147.24, -74.695, -32.684, 65.101, 36.625, -59.956]
  MoveL 10546 to (240.76, 149.6, 144.49) mm, rotated rx 180 ry 0 rz 180 deg; joints [-147.24, -74.695, -32.684, 65.101, 36.625, -59.956]
  Call Extruder(649.29886)
  MoveL 10547 to (240.71, 149.91, 144.49) mm, rotated rx 180 ry 0 rz 180 deg; joints [-147.214, -74.719, -32.637, 65.15, 36.637, -60.009]
  MoveL 10548 to (240.71, 149.91, 144.49) mm, rotated rx 180 ry 0 rz 180 deg; joints [-147.214, -74.719, -32.637, 65.15, 36.637, -60.009]
  Call Extruder(649.45987)
  MoveL 10549 to (240.66, 150.21, 144.49) mm, rotated rx -180 ry 0 rz 180 deg; joints [-147.189, -74.742, -32.589, 65.2, 36.65, -60.062]
  MoveL 10550 to (240.66, 150.21, 144.49) mm, rotated rx -180 ry 0 rz 180 deg; joints [-147.189, -74.742, -32.589, 65.2, 36.65, -60.062]
  Call Extruder(649.62162)
  MoveL 10551 to (240.61, 150.52, 144.49) mm, rotated rx -180 ry 0 rz -180 deg; joints [-147.163, -74.767, -32.542, 65.25, 36.662, -60.115]
  MoveL 10552 to (240.61, 150.52, 144.49) mm, rotated rx -180 ry 0 rz -180 deg; joints [-147.163, -74.767, -32.542, 65.25, 36.662, -60.115]
  Call Extruder(649.78409)
  MoveL 10553 to (240.56, 150.83, 144.49) mm, rotated rx 180 ry 0 rz -180 deg; joints [-147.138, -74.791, -32.494, 65.3, 36.674, -60.167]
  MoveL 10554 to (240.56, 150.83, 144.49) mm, rotated rx 180 ry 0 rz -180 deg; joints [-147.138, -74.791, -32.494, 65.3, 36.674, -60.167]
  Call Extruder(649.91802)
  MoveL 10555 to (240.52, 151.07, 144.49) mm, rotated rx 180 ry 0 rz 180 deg; joints [-147.117, -74.809, -32.458, 65.34, 36.685, -60.209]
  MoveL 10556 to (240.52, 151.07, 144.49) mm, rotated rx 180 ry 0 rz 180 deg; joints [-147.117, -74.809, -32.458, 65.34, 36.685, -60.209]
  Call Extruder(650.05255)
  MoveL 10557 to (240.47, 151.32, 144.49) mm, rotated rx -180 ry 0 rz -180 deg; joints [-147.095, -74.827, -32.423, 65.379, 36.696, -60.249]
  MoveL 10558 to (240.47, 151.32, 144.49) mm, rotated rx -180 ry 0 rz -180 deg; joints [-147.095, -74.827, -32.423, 65.379, 36.696, -60.249]
  Call Extruder(650.18770)
  MoveL 10559 to (240.42, 151.57, 144.49) mm, rotated rx -180 ry 0 rz 180 deg; joints [-147.074, -74.845, -32.387, 65.418, 36.707, -60.29]
  MoveL 10560 to (240.42, 151.57, 144.49) mm, rotated rx -180 ry 0 rz 180 deg; joints [-147.074, -74.845, -32.387, 65.418, 36.707, -60.29]
  Call Extruder(650.32346)
  MoveL 10561 to (240.37, 151.82, 144.49) mm, rotated rx -180 ry 0 rz -180 deg; joints [-147.053, -74.863, -32.351, 65.457, 36.718, -60.332]
  MoveL 10562 to (240.37, 151.82, 144.49) mm, rotated rx -180 ry 0 rz -180 deg; joints [-147.053, -74.863, -32.351, 65.457, 36.718, -60.332]
  Call Extruder(650.45983)
  MoveL 10563 to (240.32, 152.07, 144.49) mm, rotated rx 180 ry 0 rz 180 deg; joints [-147.032, -74.881, -32.315, 65.496, 36.73, -60.372]
  MoveL 10564 to (240.32, 152.07, 144.49) mm, rotated rx 180 ry 0 rz 180 deg; joints [-147.032, -74.881, -32.315, 65.496, 36.73, -60.372]
  Call Extruder(650.59680)
  MoveL 10565 to (240.27, 152.32, 144.49) mm, rotated rx 180 ry 0 rz -180 deg; joints [-147.011, -74.899, -32.279, 65.535, 36.741, -60.414]
  MoveL 10566 to (240.27, 152.32, 144.49) mm, rotated rx 180 ry 0 rz -180 deg; joints [-147.011, -74.899, -32.279, 65.535, 36.741, -60.414]
  Call Extruder(650.73439)
  MoveL 10567 to (240.22, 152.57, 144.49) mm, rotated rx -180 ry 0 rz 180 deg; joints [-146.989, -74.917, -32.243, 65.575, 36.752, -60.455]
  MoveL 10568 to (240.22, 152.57, 144.49) mm, rotated rx -180 ry 0 rz 180 deg; joints [-146.989, -74.917, -32.243, 65.575, 36.752, -60.455]
  Call Extruder(650.84809)
  MoveL 10569 to (240.17, 152.77, 144.49) mm, rotated rx -180 ry 0 rz 180 deg; joints [-146.972, -74.932, -32.215, 65.606, 36.761, -60.488]
  MoveL 10570 to (240.17, 152.77, 144.49) mm, rotated rx -180 ry 0 rz 180 deg; joints [-146.972, -74.932, -32.215, 65.606, 36.761, -60.488]
  Call Extruder(650.96224)
  MoveL 10571 to (240.13, 152.98, 144.49) mm, rotated rx 180 ry 0 rz -180 deg; joints [-146.954, -74.946, -32.187, 65.638, 36.771, -60.521]
  MoveL 10572 to (240.13, 152.98, 144.49) mm, rotated rx 180 ry 0 rz -180 deg; joints [-146.954, -74.946, -32.187, 65.638, 36.771, -60.521]
  Call Extruder(651.07684)
  MoveL 10573 to (240.08, 153.18, 144.49) mm, rotated rx 180 ry 0 rz 180 deg; joints [-146.937, -74.96, -32.158, 65.669, 36.78, -60.553]
  MoveL 10574 to (240.08, 153.18, 144.49) mm, rotated rx 180 ry 0 rz 180 deg; joints [-146.937, -74.96, -32.158, 65.669, 36.78, -60.553]
  Call Extruder(651.19190)
  MoveL 10575 to (240.04, 153.39, 144.49) mm, rotated rx 180 ry 0 rz -180 deg; joints [-146.919, -74.975, -32.13, 65.701, 36.79, -60.586]
  MoveL 10576 to (240.04, 153.39, 144.49) mm, rotated rx 180 ry 0 rz -180 deg; joints [-146.919, -74.975, -32.13, 65.701, 36.79, -60.586]
  Call Extruder(651.31412)
  MoveL 10577 to (239.98, 153.6, 144.49) mm, rotated rx 180 ry 0 rz 180 deg; joints [-146.9, -74.988, -32.103, 65.732, 36.801, -60.619]
  MoveL 10578 to (239.98, 153.6, 144.49) mm, rotated rx 180 ry 0 rz 180 deg; joints [-146.9, -74.988, -32.103, 65.732, 36.801, -60.619]
  Call Extruder(651.44378)
  MoveL 10579 to (239.92, 153.82, 144.49) mm, rotated rx 180 ry 0 rz -180 deg; joints [-146.88, -75.001, -32.078, 65.764, 36.813, -60.651]
  MoveL 10580 to (239.92, 153.82, 144.49) mm, rotated rx 180 ry 0 rz -180 deg; joints [-146.88, -75.001, -32.078, 65.764, 36.813, -60.651]
  Call Extruder(651.57401)
  MoveL 10581 to (239.85, 154.05, 144.49) mm, rotated rx 180 ry 0 rz 180 deg; joints [-146.86, -75.014, -32.053, 65.795, 36.825, -60.683]
  MoveL 10582 to (239.85, 154.05, 144.49) mm, rotated rx 180 ry 0 rz 180 deg; joints [-146.86, -75.014, -32.053, 65.795, 36.825, -60.683]
  Call Extruder(651.70480)
  MoveL 10583 to (239.78, 154.27, 144.49) mm, rotated rx 180 ry 0 rz -180 deg; joints [-146.84, -75.027, -32.027, 65.827, 36.838, -60.715]
  MoveL 10584 to (239.78, 154.27, 144.49) mm, rotated rx 180 ry 0 rz -180 deg; joints [-146.84, -75.027, -32.027, 65.827, 36.838, -60.715]
  Call Extruder(651.83615)
  MoveL 10585 to (239.71, 154.49, 144.49) mm, rotated rx 180 ry 0 rz 180 deg; joints [-146.82, -75.039, -32.002, 65.859, 36.85, -60.747]
  MoveL 10586 to (239.71, 154.49, 144.49) mm, rotated rx 180 ry 0 rz 180 deg; joints [-146.82, -75.039, -32.002, 65.859, 36.85, -60.747]
  Call Extruder(651.94805)
  MoveL 10587 to (239.65, 154.68, 144.49) mm, rotated rx -180 ry 0 rz 180 deg; joints [-146.803, -75.049, -31.982, 65.885, 36.861, -60.774]
  MoveL 10588 to (239.65, 154.68, 144.49) mm, rotated rx -180 ry 0 rz 180 deg; joints [-146.803, -75.049, -31.982, 65.885, 36.861, -60.774]
  Call Extruder(652.06040)
  MoveL 10589 to (239.59, 154.87, 144.49) mm, rotated rx 180 ry 0 rz 180 deg; joints [-146.785, -75.06, -31.962, 65.911, 36.872, -60.8]
  MoveL 10590 to (239.59, 154.87, 144.49) mm, rotated rx 180 ry 0 rz 180 deg; joints [-146.785, -75.06, -31.962, 65.911, 36.872, -60.8]
  Call Extruder(652.17319)
  MoveL 10591 to (239.53, 155.06, 144.49) mm, rotated rx 180 ry 0 rz 180 deg; joints [-146.768, -75.07, -31.942, 65.937, 36.883, -60.826]
  MoveL 10592 to (239.53, 155.06, 144.49) mm, rotated rx 180 ry 0 rz 180 deg; joints [-146.768, -75.07, -31.942, 65.937, 36.883, -60.826]
  Call Extruder(652.28642)
  MoveL 10593 to (239.47, 155.25, 144.49) mm, rotated rx 180 ry 0 rz -180 deg; joints [-146.751, -75.08, -31.922, 65.963, 36.894, -60.852]
  MoveL 10594 to (239.47, 155.25, 144.49) mm, rotated rx 180 ry 0 rz -180 deg; joints [-146.751, -75.08, -31.922, 65.963, 36.894, -60.852]
  Call Extruder(652.40010)
  MoveL 10595 to (239.41, 155.44, 144.49) mm, rotated rx -180 ry 0 rz 180 deg; joints [-146.734, -75.09, -31.902, 65.989, 36.905, -60.879]
  MoveL 10596 to (239.41, 155.44, 144.49) mm, rotated rx -180 ry 0 rz 180 deg; joints [-146.734, -75.09, -31.902, 65.989, 36.905, -60.879]
  Call Extruder(652.58206)
  MoveL 10597 to (239.29, 155.73, 144.49) mm, rotated rx 180 ry 0 rz -180 deg; joints [-146.706, -75.102, -31.879, 66.025, 36.925, -60.914]
  MoveL 10598 to (239.29, 155.73, 144.49) mm, rotated rx 180 ry 0 rz -180 deg; joints [-146.706, -75.102, -31.879, 66.025, 36.925, -60.914]
  Call Extruder(652.76478)
  MoveL 10599 to (239.17, 156.02, 144.49) mm, rotated rx 180 ry 0 rz 180 deg; joints [-146.678, -75.113, -31.856, 66.061, 36.945, -60.949]
  MoveL 10600 to (239.17, 156.02, 144.49) mm, rotated rx 180 ry 0 rz 180 deg; joints [-146.678, -75.113, -31.856, 66.061, 36.945, -60.949]
  Call Extruder(652.93520)
  MoveL 10601 to (239.05, 156.29, 144.49) mm, rotated rx -180 ry 0 rz 180 deg; joints [-146.652, -75.124, -31.836, 66.095, 36.963, -60.981]
  MoveL 10602 to (239.05, 156.29, 144.49) mm, rotated rx -180 ry 0 rz 180 deg; joints [-146.652, -75.124, -31.836, 66.095, 36.963, -60.981]
  Call Extruder(653.09321)
  MoveL 10603 to (238.94, 156.54, 144.49) mm, rotated rx 180 ry 0 rz 180 deg; joints [-146.628, -75.133, -31.817, 66.125, 36.98, -61.01]
  MoveL 10604 to (238.94, 156.54, 144.49) mm, rotated rx 180 ry 0 rz 180 deg; joints [-146.628, -75.133, -31.817, 66.125, 36.98, -61.01]
  Call Extruder(653.25183)
  MoveL 10605 to (238.84, 156.79, 144.49) mm, rotated rx -180 ry 0 rz 180 deg; joints [-146.604, -75.142, -31.799, 66.155, 36.998, -61.04]
  MoveL 10606 to (238.84, 156.79, 144.49) mm, rotated rx -180 ry 0 rz 180 deg; joints [-146.604, -75.142, -31.799, 66.155, 36.998, -61.04]
  Call Extruder(653.45800)
  MoveL 10607 to (238.66, 157.09, 144.49) mm, rotated rx -180 ry 0 rz 180 deg; joints [-146.573, -75.146, -31.79, 66.186, 37.023, -61.066]
  MoveL 10608 to (238.66, 157.09, 144.49) mm, rotated rx -180 ry 0 rz 180 deg; joints [-146.573, -75.146, -31.79, 66.186, 37.023, -61.066]
  Call Extruder(653.66494)
  MoveL 10609 to (238.49, 157.4, 144.49) mm, rotated rx -180 ry 0 rz -180 deg; joints [-146.542, -75.15, -31.782, 66.216, 37.049, -61.092]
  MoveL 10610 to (238.49, 157.4, 144.49) mm, rotated rx -180 ry 0 rz -180 deg; joints [-146.542, -75.15, -31.782, 66.216, 37.049, -61.092]
  Call Extruder(653.87267)
  MoveL 10611 to (238.31, 157.7, 144.49) mm, rotated rx -180 ry 0 rz -180 deg; joints [-146.51, -75.155, -31.774, 66.246, 37.075, -61.119]
  MoveL 10612 to (238.31, 157.7, 144.49) mm, rotated rx -180 ry 0 rz -180 deg; joints [-146.51, -75.155, -31.774, 66.246, 37.075, -61.119]
  Call Extruder(654.08118)
  MoveL 10613 to (238.13, 158.01, 144.49) mm, rotated rx 180 ry 0 rz 180 deg; joints [-146.479, -75.159, -31.766, 66.276, 37.101, -61.145]
  MoveL 10614 to (238.13, 158.01, 144.49) mm, rotated rx 180 ry 0 rz 180 deg; joints [-146.479, -75.159, -31.766, 66.276, 37.101, -61.145]
  Call Extruder(654.26072)
  MoveL 10615 to (237.96, 158.25, 144.49) mm, rotated rx 180 ry 0 rz 180 deg; joints [-146.452, -75.157, -31.77, 66.295, 37.126, -61.159]
  MoveL 10616 to (237.96, 158.25, 144.49) mm, rotated rx 180 ry 0 rz 180 deg; joints [-146.452, -75.157, -31.77, 66.295, 37.126, -61.159]
  Call Extruder(654.59412)
  MoveL 10617 to (237.63, 158.7, 144.49) mm, rotated rx -180 ry 0 rz 180 deg; joints [-146.402, -75.152, -31.779, 66.329, 37.171, -61.184]
  MoveL 10618 to (237.63, 158.7, 144.49) mm, rotated rx -180 ry 0 rz 180 deg; joints [-146.402, -75.152, -31.779, 66.329, 37.171, -61.184]
  Call Extruder(654.92872)
  MoveL 10619 to (237.3, 159.15, 144.49) mm, rotated rx -180 ry 0 rz 180 deg; joints [-146.352, -75.147, -31.788, 66.364, 37.217, -61.209]
  Call Extruder(655.75669)
  MoveL 10620 to (236.39, 160.19, 144.49) mm, rotated rx 180 ry 0 rz 180 deg; joints [-146.229, -75.112, -31.859, 66.419, 37.338, -61.233]
  Call Extruder(656.58460)
  MoveL 10621 to (235.35, 161.1, 144.49) mm, rotated rx -180 ry 0 rz 180 deg; joints [-146.109, -75.043, -31.995, 66.433, 37.47, -61.207]
  Call Extruder(656.75191)
  MoveL 10622 to (235.13, 161.27, 144.49) mm, rotated rx 180 ry 0 rz 180 deg; joints [-146.086, -75.024, -32.032, 66.43, 37.498, -61.194]
  MoveL 10623 to (235.13, 161.27, 144.49) mm, rotated rx 180 ry 0 rz 180 deg; joints [-146.086, -75.024, -32.032, 66.43, 37.498, -61.194]
  Call Extruder(657.08534)
  MoveL 10624 to (234.68, 161.59, 144.49) mm, rotated rx -180 ry 0 rz 180 deg; joints [-146.039, -74.987, -32.106, 66.424, 37.554, -61.169]
  MoveL 10625 to (234.68, 161.59, 144.49) mm, rotated rx -180 ry 0 rz 180 deg; joints [-146.039, -74.987, -32.106, 66.424, 37.554, -61.169]
  Call Extruder(657.41758)
  MoveL 10626 to (234.22, 161.92, 144.49) mm, rotated rx 180 ry 0 rz 180 deg; joints [-145.992, -74.95, -32.179, 66.418, 37.61, -61.144]
  MoveL 10627 to (234.22, 161.92, 144.49) mm, rotated rx 180 ry 0 rz 180 deg; joints [-145.992, -74.95, -32.179, 66.418, 37.61, -61.144]
  Call Extruder(657.53524)
  MoveL 10628 to (234.05, 162.02, 144.49) mm, rotated rx 180 ry 0 rz 180 deg; joints [-145.976, -74.933, -32.212, 66.411, 37.63, -61.13]
